// TwinCAT 3 PLC project Unbenannt1
// Title: Sample PackML_V2
// Company: Beckhoff Automation GmbH
// Author: Beckhoff Automation GmbH
// ProjectVersion: 3.0.3.0
// Description: Sample PackML_V2
// ProgramVersion: 3.1.4026.16
// libraries:
//   Tc2_MC2, * (Beckhoff Automation GmbH)
//   Tc2_Standard, * (Beckhoff Automation GmbH)
//   Tc2_System, * (Beckhoff Automation GmbH)
//   Tc2_Utilities, * (Beckhoff Automation GmbH)
//   Tc3_Analytics, * (Beckhoff Automation GmbH)
//   Tc3_Module, * (Beckhoff Automation GmbH)
//   Tc3_PackML_V2, * (Beckhoff Automation GmbH)
//   VisuDialogs, * (System)
// project tree:
//   DUTs/ E_PMLUserUnitMode.TcDUT, E_UnitName.TcDUT, ST_AxFunctions.TcDUT, ST_AxFunctionsAdmin.TcDUT, ST_ChangeIntoProduction.TcDUT, ST_AxFunctionsPTP.TcDUT, ST_UnitInfo.TcDUT
//   / GlobalTextList.TcGTLO, PlcTask.TcTTO, Visualization Manager.TcVMO (not stored)
//   GVLs/ GlobalVariables.TcGVL
//   POUs/General/ FB_AxisGeneral.TcPOU, FB_Cylinder.TcPOU, FB_Generic.TcPOU, FB_Velocity.TcPOU, FB_Visu.TcPOU, Ton_Break.TcPOU
//   POUs/ MAIN.TcPOU
//   POUs/Units/Conveyor/ FB_AxisMain.TcPOU
//   POUs/Units/Ejection/ FB_AxixEjection.TcPOU, FB_Ejector.TcPOU, FB_Sensor.TcPOU
//   POUs/Units/Machine/ FB_Machine.TcPOU
//   POUs/Units/Seperation/ FB_Seperation.TcPOU
//   Version/ Global_Version.TcGVL
//   VISUs/Templates/ VIS_TemplateCommand.TcVIS, VIS_TemplateKeys.TcVIS, VIS_TemplateMachine.TcVIS, VIS_TemplatePMLStateModel.TcVIS, VIS_TemplateToProduction.TcVIS
//   VISUs/ VIS_Main.TcVIS
// real-time tasks:
//   TASK PlcTask: cycle T#10ms, priority 20, ADS port 350
//   TASK PlcTask1: cycle T#10ms, priority 21, ADS port 351
//   TASK AnalyticsTask: cycle T#10ms, priority 1, ADS port 352
//   TASK AnalyticsTask_C1: cycle T#10ms, priority 22, ADS port 353
// motion (NC):
//   TASK NC-Task 1 SAF: cycle T#2ms, priority 4, ADS port 501
//   TASK NC-Task 1 SVB: cycle T#10ms, priority 8, ADS port 511
//   AXIS Axis 1 - Main Belt (id 1)
//     OtherSettings: AllowMotionCmdToSlave=true
//     encoder EncType=1
//     drive DrvType=5
//       TimeComp: TaskDelayCycles=1
//     controller CtrType=1
//       CtrPara: PriorControlFactor=1
//         Observer: BandWidth=20
//   AXIS Axis 2 - Metal Belt (id 2)
//     OtherSettings: AllowMotionCmdToSlave=true
//     encoder EncType=1
//     drive DrvType=5
//       TimeComp: TaskDelayCycles=1
//     controller CtrType=1
//       CtrPara: PriorControlFactor=1
//         Observer: BandWidth=20
//   AXIS Axis 3 - Plastic Belt (id 3)
//     OtherSettings: AllowMotionCmdToSlave=true
//     encoder EncType=1
//     drive DrvType=5
//       TimeComp: TaskDelayCycles=1
//     controller CtrType=1
//       CtrPara: PriorControlFactor=1
//         Observer: BandWidth=20
// variable links:
//   Unbenannt1/Unbenannt1 Instance <-> NC-Task 1 SAF/Axes/Axis 1 - Main Belt
//     PlcTask Inputs/GlobalVariables.AxisMain.NcToPlc <-> Outputs/ToPlc
//     PlcTask Outputs/GlobalVariables.AxisMain.PlcToNc <-> Inputs/FromPlc
//   Unbenannt1/Unbenannt1 Instance <-> NC-Task 1 SAF/Axes/Axis 2 - Metal Belt
//     PlcTask Inputs/GlobalVariables.AxisMetal.NcToPlc <-> Outputs/ToPlc
//     PlcTask Outputs/GlobalVariables.AxisMetal.PlcToNc <-> Inputs/FromPlc
//   Unbenannt1/Unbenannt1 Instance <-> NC-Task 1 SAF/Axes/Axis 3 - Plastic Belt
//     PlcTask Inputs/GlobalVariables.AxisPlastic.NcToPlc <-> Outputs/ToPlc
//     PlcTask Outputs/GlobalVariables.AxisPlastic.PlcToNc <-> Inputs/FromPlc
//   Unbenannt1/Unbenannt1 Instance <-> Unbenannt1/Unbenannt1 Instance
//     PlcTask Inputs/MAIN.fbMachine.fbEjectionMetal.bSensorEjection <-> PlcTask Outputs/MAIN.fbVisu.bMetalSensor
//     PlcTask Inputs/MAIN.fbMachine.fbEjectionMetal.fbCylinderEjection.bAtBasePos <-> PlcTask Outputs/MAIN.fbVisu.bMetalAtBase
//     PlcTask Inputs/MAIN.fbMachine.fbEjectionMetal.fbCylinderEjection.bAtWorkPos <-> PlcTask Outputs/MAIN.fbVisu.bMetalAtWork
//     PlcTask Inputs/MAIN.fbMachine.fbEjectionPlastic.bSensorEjection <-> PlcTask Outputs/MAIN.fbVisu.bPlasticSensor
//     PlcTask Inputs/MAIN.fbMachine.fbEjectionPlastic.fbCylinderEjection.bAtBasePos <-> PlcTask Outputs/MAIN.fbVisu.bPlasticAtBase
//     PlcTask Inputs/MAIN.fbMachine.fbEjectionPlastic.fbCylinderEjection.bAtWorkPos <-> PlcTask Outputs/MAIN.fbVisu.bPlasticAtWork
//     PlcTask Inputs/MAIN.fbMachine.fbSeperation.bSensorBarrier <-> PlcTask Outputs/MAIN.fbVisu.bBarrierSensor
//     PlcTask Inputs/MAIN.fbMachine.fbSeperation.fbCylinderBarrier.bAtBasePos <-> PlcTask Outputs/MAIN.fbVisu.bBarrierAtBase
//     PlcTask Inputs/MAIN.fbMachine.fbSeperation.fbCylinderBarrier.bAtWorkPos <-> PlcTask Outputs/MAIN.fbVisu.bBarrierAtWork
//     PlcTask Inputs/MAIN.fbMachine.fbSeperation.fbCylinderClamb.bAtBasePos <-> PlcTask Outputs/MAIN.fbVisu.bClampAtBase
//     PlcTask Inputs/MAIN.fbMachine.fbSeperation.fbCylinderClamb.bAtWorkPos <-> PlcTask Outputs/MAIN.fbVisu.bClampAtWork

CONFIGURATION Unbenannt1
    RESOURCE PLC ON TwinCAT3
        TASK PlcTask(INTERVAL := T#10ms, PRIORITY := 20);
        PROGRAM MAIN WITH PlcTask : MAIN;
    END_RESOURCE
END_CONFIGURATION

// ---- DUTs/E_PMLUserUnitMode.TcDUT
//Enumeration for User Modes
TYPE E_PMLUserUnitMode : (
	ePMLUnitMode_Service		:=  4,
	ePMLUnitMode_Usermode2		:=  5,
	ePMLUnitMode_Usermode3		:=  6,
	ePMLUnitMode_Usermode4		:=  7,
	ePMLUnitMode_Usermode5 		:=  8,
	ePMLUnitMode_Usermode6 		:=  9,
	ePMLUnitMode_Usermode7 		:=  10
) DINT;
END_TYPE

// ---- DUTs/E_UnitName.TcDUT
//Enumeration for Machineunits
TYPE E_UnitName :
(
	eMachine		:= 1,
	eSeperation		:= 2,
	eEjectorPlastic	:= 3,
	eAxisMain		:= 4,
	eEjectorMetal	:= 5,
	eSensorPlastic	:= 6,
	eAxisPlastic	:= 7,
	eSensorMetal	:= 8,
	eAxisMetal		:= 9
)DINT;
END_TYPE

// ---- DUTs/ST_AxFunctions.TcDUT
//structure includes structures with TC Motion functions
TYPE ST_AxFunctions :
STRUCT
	Admin				: ST_AxFunctionsAdmin;
	PTP					: ST_AxFunctionsPTP;
END_STRUCT
END_TYPE

// ---- DUTs/ST_AxFunctionsAdmin.TcDUT
//structure includes axisfunctions
TYPE ST_AxFunctionsAdmin :
STRUCT
	Power	: MC_Power;
	Reset	: MC_Reset;
END_STRUCT
END_TYPE

// ---- DUTs/ST_ChangeIntoProduction.TcDUT
//structure for a visu userwindow, to chnage into productionmode
TYPE ST_ChangeIntoProduction :
STRUCT
	bYes		: BOOL;
	bNo			: BOOL;
	bYesReset	: BOOL;
END_STRUCT
END_TYPE

// ---- DUTs/ST_AxFunctionsPTP.TcDUT
//structure includes point-to-point-functions
TYPE ST_AxFunctionsPTP :
STRUCT
	MoveVelocitiy		: MC_MoveVelocity;
	MoveAbsolute1		: MC_MoveAbsolute;
	MoveAbsolute2		: MC_MoveAbsolute;
	Stop				: MC_Stop;
	Halt				: MC_Halt;
END_STRUCT
END_TYPE

// ---- DUTs/ST_UnitInfo.TcDUT
//structure includes unit information
TYPE ST_UnitInfo :
STRUCT
	Name		: STRING;
	ActState	: E_PMLState;
	ActMode		: DINT;
END_STRUCT
END_TYPE

// ---- GVLs/GlobalVariables.TcGVL
VAR_GLOBAL
		AxisMain					: AXIS_REF;						//Main belt
		AxisPlastic					: AXIS_REF;						//Plastic belt
		AxisMetal					: AXIS_REF;						//Metal belt

		bAxisMainResetDone			: BOOL;							//True if main belt ressetting is finished 
		bPlasticEjectionResetDone	: BOOL;							//True if plasticejection ressetting is finished 
		bMetalEjectionResetDone		: BOOL;							//True if metalejection ressetting is finished 
		
		PackTags					: ST_PackMLv30;					//PackTags
		
		//analytics testing//2.1
		{attribute 'TcAnalytics'}
		nVisuProductCommand			: DINT:=1512000;							//Schedule products to produce

		bButtonProductionReq		: BOOL;							//TRUE when a mode change to PRODUCTION is requested
		stChangeIntoProduction		: ST_ChangeIntoProduction;		//Result of command box "Change to Production requested"

		aUnitInfo					: ARRAY [1..12] OF ST_UnitInfo;	//Array includes the states and modes of machineunits	
		aCaption					: ARRAY [1..12] OF STRING := ['F1','F2','F3','F4','F5','F6','F7','F8','F9','F10','F11','F12'];
		aKeyPressed					: ARRAY [1..12] OF BOOL;	
		
		
		uScheduleTime	 			: ULINT	:= 2 ;//for OEE 
		//analytics testing//2.1//3600000000000
		{attribute 'TcAnalytics'}			
		lScheduledTime 				: LINT	:= 3600000000000;//1 hours=1×60×60×1,000,000,000=3,600,000,000,000 nanoseconds
		
		//analytics testing//2.1
		{attribute 'TcAnalytics'}
		uDefectiveCount 			: ULINT	:= 0 ;//for OEE 
		
		//analytics testing//2.1
		{attribute 'TcAnalytics'}
		uTotalCount 				: ULINT	:= 0 ;//for OEE 
		
		//analytics testing//2.1
		{attribute 'TcAnalytics'}
		uPlasticCount 	 			: ULINT	:= 0 ;//for plastic items 
		
		//analytics testing//2.1
		{attribute 'TcAnalytics'}
		uMetalCount 	 			: ULINT	:= 0 ;//for metal items 
		
		//analytics testing//2.1
		{attribute 'TcAnalytics'}
		bScheduleDownTime 			: BOOL	:= FALSE ;//if under maintanance mode will be under this categories
		//analytics testing//2.1
		{attribute 'TcAnalytics'}
		bUnscheduleDownTime			: BOOL	:= FALSE ;//else if under manual mode or unknown will be under this categories
		
		//analytics testing//2.1
		{attribute 'TcAnalytics'}
		bProductionMode				: BOOL	:= FALSE ;//else if under manual mode or unknown will be under this categories
		
		//analytics testing//2.2
		{attribute 'TcAnalytics'}
		lStartTime 					: LWORD	:= 3600000000000 ;//Productivity internal
		//analytics testing//2.2
		{attribute 'TcAnalytics'}
		lStopTime 					: LWORD	:= 7200000000000 ;//Productivity internal
		
		//analytics testing//2.2
		{attribute 'TcAnalytics'}
		bConfigure 					: BOOL := TRUE;//Productivity internal
		
		{attribute 'TcAnalytics'}
		bReset	 					: BOOL := FALSE;//Productivity internal
		{attribute 'TcAnalytics'}
		bTest	 					: BOOL :=FALSE;//Productivity internal
END_VAR

// ---- Version/Global_Version.TcGVL
{attribute 'TcGenerated'}
{attribute 'no-analysis'}
{attribute 'linkalways'}
// This function has been automatically generated from the project information.
VAR_GLOBAL CONSTANT
	{attribute 'const_non_replaced'}
	stLibVersion_Sample_PackML_V2 : ST_LibVersion := (iMajor := 3, iMinor := 0, iBuild := 3, iRevision := 0, nFlags := 1, sVersion := '3.0.3.0');
END_VAR

// ---- POUs/MAIN.TcPOU
// Disclaimer
// 
// This publication contains statements about the suitability of our products for certain areas of application. These statements are based on typical features of our products. The examples shown in this publication are for demonstration purposes only. 
// The information provided herein should not be regarded as specific operation characteristics. It is incumbent on the customer to check and decide whether a product is suitable for use in a particular application. 
// We do not give any warranty that the source code which is made available with this publication is complete or accurate. 
//
// THE SAMPLE CODE CONTAINED IN THIS PUBLICATION IS PROVIDED “AS IS” WITHOUT WARRANTY OF ANY KIND, EITHER EXPRESSED, IMPLIED OR STATUTORY, INCLUDING WITHOUT LIMITATION, ANY WARRANTY WITH RESPECT TO NON-INFRINGEMENT, FREEDOM FROM PROPRIETARY RIGHTS OF THIRD PARTIES OR FITNESS FOR ANY PARTICULAR PURPOSE. 
// This publication may be changed from time to time without prior notice. No liability is assumed for errors and/or omissions. Our products are described in detail in our data sheets and documentations. Product-specific warnings and cautions must be observed. 
// For the latest version of our data sheets and documentations visit our website (www.beckhoff.de). 
//
// © Beckhoff Automation GmbH & Co. KG, 2022
// The reproduction, distribution and utilization of this document as well as the communication of its contents to others without express authorization is prohibited. Offenders will be held liable for the payment of damages. All rights reserved in the event of the grant of a patent, utility model or design.
PROGRAM MAIN
VAR_INPUT
	bExecuteComplete			: BOOL;									//Command Execute Complete, not defined
END_VAR
VAR
	UserModeCofig				: PML_UnitModeConfig;					//User can configure his own Mode
	
	fbMachine					: FB_Machine;							//Instance of FB_Machine
	bMachineStartedUp			: BOOL := FALSE;						//TRUE, when first PLC-Cycle finish

	fbVisu						: FB_Visu;								//Visualization
	
	fbTrigger					: F_TRIG;								//Trigger for resseting Counters

	fbLocalSystemTime			 : FB_LocalSystemTime;					//Get local Systemtime
	
	fbTriggerErrorMainAxis		: R_TRIG;								//Trigger for detecting Error on Mainaxis and write into PackTags
	fbTriggerErrorMetalAxis		: R_TRIG;								//Trigger for detecting Error on Metalaxis and write into PackTags
	fbTriggerErrorPlasticAxis	: R_TRIG;								//Trigger for detecting Error on Plasticaxis and write into PackTags
	
	nStateCommandCheck			: DINT;									//State to handle with statecommands
	//OEE UI
	todStart     				: TIME_OF_DAY:= TOD#00:00:00.000000000; // 8 AM
	//todStart     				: DT:=DT#2025-06-30-13:55:00;
	////todStart     				:  TIME := TIME#14H;
	//OEE UI
	todStop     				: TIME_OF_DAY:=TOD#09:00:00.000000000; // 5 PM
	//todStop     				: DT:=DT#2025-06-30-14:00:00;
	////todStop     				:  TIME := TIME#16H;

  	iLocalCount					: DINT;

	bTest1	:	BOOL;
	Test1	: TON;
END_VAR

//Configure Usermode 1
A_UnitModeConfig();

//Runs the first PLC-Cycle
IF fbMachine.bUndefinedDone AND NOT bMachineStartedUp THEN
	PackTags.Command.CntrlCmd	:= ePMLCommand_Abort;
	bMachineStartedUp			:= TRUE;
END_IF

M_SetPackTags();
M_SetPackTagsErrorWarning();

bButtonProductionReq := PackTags.Command.UnitMode = ePMLProtUnitMode_Production AND PackTags.Status.UnitModeCurrent <> PackTags.Command.UnitMode;

//Checking the Statecommands
CASE nStateCommandCheck OF
0:
	IF NOT (AxisMain.Status.Error OR AxisPlastic.Status.Error OR AxisMetal.Status.Error) THEN
		nStateCommandCheck:= 1;
	ELSE
		nStateCommandCheck:= 2;
	END_IF
1:
	IF PackTags.Command.CntrlCmd = ePMLCommand_Clear		
	  AND fbMachine.eState = ePMLState_Aborted	THEN
			fbMachine.eCommand	:= ePMLCommand_Clear;
	ELSIF PackTags.Command.CntrlCmd = ePMLCommand_Reset		
	  AND (fbMachine.eState = ePMLState_Stopped OR fbMachine.eState = ePMLState_Complete) THEN
			fbMachine.eCommand	:= ePMLCommand_Reset;
	ELSIF PackTags.Command.CntrlCmd = ePMLCommand_Start	
	  AND (fbMachine.eState = ePMLState_Idle OR (stPMLUnitModeConfiguration[fbMachine.eMode].aStateDisabled[ePMLState_Idle] AND fbMachine.eState = ePMLState_Stopped))
	  AND (NOT (PackTags.Command.Parameter[2].Value <= 0) OR NOT (fbMachine.eMode = 1))THEN
			fbMachine.eCommand	:= ePMLCommand_Start; 
	ELSIF PackTags.Command.CntrlCmd = ePMLCommand_Hold		
	  AND fbMachine.eState = ePMLState_Execute	
	  AND( fbMachine.eMode =  1 OR fbMachine.eMode =  4 OR fbMachine.eMode = 2)  THEN
			 fbMachine.eCommand	:= ePMLCommand_Hold;
	ELSIF PackTags.Command.CntrlCmd = ePMLCommand_Suspend	
	  AND fbMachine.eState = ePMLState_Execute	
	  AND (fbMachine.eMode = 4 OR fbMachine.eMode = 1)THEN
			 fbMachine.eCommand	:= ePMLCommand_Suspend;
	ELSIF PackTags.Command.CntrlCmd = ePMLCommand_Unhold	
	  AND fbMachine.eState = ePMLState_Held		THEN
			 fbMachine.eCommand	:= ePMLCommand_Unhold;
	ELSIF PackTags.Command.CntrlCmd = ePMLCommand_Unsuspend	
	  AND fbMachine.eState = ePMLState_Suspended	THEN
			 fbMachine.eCommand	:= ePMLCommand_Unsuspend;
	ELSIF PackTags.Command.CntrlCmd = ePMLCommand_Abort	THEN
			fbMachine.eCommand	:= ePMLCommand_Abort;
	ELSIF PackTags.Command.CntrlCmd = ePMLCommand_Stop	THEN
			fbMachine.eCommand	:= ePMLCommand_Stop;
	END_IF
	nStateCommandCheck:=0;
	
2:
	fbMachine.eCommand	:= ePMLCommand_Abort;
	IF fbMachine.eState = ePMLState_Aborted AND PackTags.Command.CntrlCmd = ePMLCommand_Clear THEN
		nStateCommandCheck:=1;
	END_IF
END_CASE

//
//Set the Packtags
M_SetPackTags();

//set the errors and warnings in Packtags
M_SetPackTagsErrorWarning();

//Call Visu
M_CallVisu();

//Call FB_Machine
fbMachine(eModeCommand:= PackTags.Command.UnitMode,  eMode => PackTags.Status.UnitModeCurrent, eState =>PackTags.Status.StateCurrent);

//for analytics conversion
lScheduledTime:= ULINT_TO_LINT(uScheduleTime*60*60*1000000000);
uTotalCount:= DINT_TO_ULINT(PackTags.Admin.ProdProcessedCount[1].Count);
uPlasticCount:= DINT_TO_ULINT(PackTags.Admin.ProdProcessedCount[3].Count);
uMetalCount:= DINT_TO_ULINT(PackTags.Admin.ProdProcessedCount[4].Count);

IF PackTags.Status.UnitModeCurrent = 1 THEN
	bProductionMode:= TRUE;
ELSE
	bProductionMode:= FALSE;
END_IF

//packml 2.2
// Convert to LWORD (100-ns ticks), then multiply
lStartTime := TO_LWORD(todStart) * 1000000;
lStopTime := TO_LWORD(todStop) * 1000000;

Test1(in:= bTest1,pt:= T#0.5S);
IF iLocalCount <> PackTags.Admin.ProdProcessedCount[1].Count THEN
	bTest:= TRUE;
	bTest1:= TRUE;
	iLocalCount := PackTags.Admin.ProdProcessedCount[1].Count;
ELSIF iLocalCount = PackTags.Admin.ProdProcessedCount[1].Count AND Test1.q THEN
	bTest:= FALSE;
	bTest1:= FALSE;
END_IF

ACTION A_UnitModeConfig:
UserModeCofig(
	eMode							:= ePMLUnitMode_Service, 
	bDisableClearing				:= TRUE, 
	bDisableStarting				:= TRUE, 
	bDisableSuspended				:= FALSE, 
	bDisableStopping				:= TRUE, 
	bDisableAborting				:= TRUE, 
	bDisableHolding					:= TRUE, 
	bDisableHeld					:= TRUE, 
	bDisableUnholding				:= TRUE, 
	bDisableSuspending				:= TRUE, 
	bDisableUnsuspending			:= TRUE, 
	bDisableResetting				:= TRUE, 
	bDisableIdle					:= TRUE, 
	bDisableCompleting				:= TRUE, 
	bDisableComplete				:= TRUE, 
	bEnableUnitModeChangeStopped	:= TRUE, 
	bEnableUnitModeChangeIdle		:= FALSE, 
	bEnableUnitModeChangeSuspended	:= FALSE, 
	bEnableUnitModeChangeExecute	:= FALSE, 
	bEnableUnitModeChangeAborted	:= TRUE, 
	bEnableUnitModeChangeHeld		:= FALSE, 
	bEnableUnitModeChangeComplete	:= FALSE, 
	bError							=> , 
	nErrorId						=> );
END_ACTION

METHOD M_CallVisu
VAR_INPUT
END_VAR
//Calling FB_Visu
fbVisu(
	fAxisVelo				:= PackTags.Command.Parameter[1].Value, 							
	bMainAxisMoves			:= AxisMain.Status.Moving, 
	bMetalAxisMoves			:= AxisMetal.Status.Moving, 
	bPlasticAxisMoves		:= AxisPlastic.Status.Moving, 
	bClampToWork			:= fbMachine.bClampToWork, 
	bBarrierToWork			:= fbMachine.bBarrierToWork, 
	bMetalToWork			:= fbMachine.bMetalToWork , 
	bPlasticToWork			:= fbMachine.bPlasticToWork ,
	bReset					:= ,
	aKeyPressed				:= aKeyPressed,
	aUnitInfo				:= aUnitInfo,
	fYClamp					=> , 
	fYBarrier				=> , 
	fYMetal					=> , 
	fYPlastic				=> , 
	bButtonPowerOut			=> , 
	bButtonMainFwOut		=> fbMachine.bButtonMainFw,  
	bButtonMetalFwOut		=> fbMachine.bButtonMetalFw, 
	bButtonPlasticFwOut		=> fbMachine.bButtonPlasticFw, 
	bButtonClampToWorkOut	=> fbMachine.bButtonClampToWork, 
	bButtonBarrierToWorkOut	=> fbMachine.bButtonBarrierToWork, 
	bButtonMetalToWorkOut	=> fbMachine.bButtonMetalToWork, 
	bButtonPlasticToWorkOut	=> fbMachine.bButtonPlasticToWork,
	bInvalidEntry			=> ,
	aCaption				=> aCaption,
	eModeVisu				=> ,
	eStateVisu				=> ,
	sUnitName				=> ,
	iFrameVisible			=> );
END_METHOD

METHOD M_SetPackTags
VAR_INPUT
END_VAR
VAR	
END_VAR
//***************************Writing Data into PackTags***************************
//Define the product metalbox 
PackTags.Command.Product[1].ProductID					:= 1;
PackTags.Command.Product[1].ProcessVariables[1].ID		:= 1;
PackTags.Command.Product[1].ProcessVariables[1].Name	:= 'CylinderPressureMetal';
PackTags.Command.Product[1].ProcessVariables[1].Unit	:= 'Bar';
PackTags.Command.Product[1].ProcessVariables[1].Value	:= 5;
(*Thre are no useful Ingrediens for Metalboxes in this Machine*)

//Define the product plasticbox
PackTags.Command.Product[2].ProductID					:= 2;
PackTags.Command.Product[2].ProcessVariables[1].ID		:= 2;
PackTags.Command.Product[2].ProcessVariables[1].Name	:= 'CylinderPressurePlastic';
PackTags.Command.Product[2].ProcessVariables[1].Unit	:= 'Bar';
PackTags.Command.Product[2].ProcessVariables[1].Value	:= 3;
(*Thre are no useful Ingrediens for Plasticboxes in this Machine*)

//Parameters for the production, here set the velocity from MainBelt
PackTags.Command.Parameter[1].ID				:= 3;
PackTags.Command.Parameter[1].Name				:= 'MainBeltVelo';
PackTags.Command.Parameter[1].Unit				:= 'mm/s';
PackTags.Command.Parameter[1].Value				:= 100.0;

//Number of producing products
PackTags.Command.Parameter[2].ID				:= 4;
PackTags.Command.Parameter[2].Name				:= 'Quantity';
PackTags.Command.Parameter[2].Unit				:= 'Box';

//Parameters for the production, here set the velocity from MetalBelt
PackTags.Command.Parameter[3].ID				:= 5;
PackTags.Command.Parameter[3].Name				:= 'MetalBeltVelo';
PackTags.Command.Parameter[3].Unit				:= 'mm/s';
PackTags.Command.Parameter[3].Value				:= 100.0;

//Parameters for the production, here set the velocity from PlasticBelt
PackTags.Command.Parameter[4].ID				:= 6;
PackTags.Command.Parameter[4].Name				:= 'PlasticBeltVelo';
PackTags.Command.Parameter[4].Unit				:= 'mm/s';
PackTags.Command.Parameter[4].Value				:= 100.0;

//Parameters for the production, here get the velocity from PlasticBelt
PackTags.Status.Parameter[1].ID					:= 7;
PackTags.Status.Parameter[1].Name				:= 'MainBeltVelo';
PackTags.Status.Parameter[1].Unit				:= 'mm/s';
PackTags.Status.Parameter[1].Value				:= LREAL_TO_REAL(AxisMain.NcToPlc.ActVelo);

//Parameters for the production, here get the velocity from PlasticBelt
PackTags.Status.Parameter[2].ID					:= 8;
PackTags.Status.Parameter[2].Name				:= 'MetalBeltVelo';
PackTags.Status.Parameter[2].Unit				:= 'mm/s';
PackTags.Status.Parameter[2].Value				:=  LREAL_TO_REAL(AxisMetal.NcToPlc.ActVelo);

//Parameters for the production, here get the velocity from PlasticBelt
PackTags.Status.Parameter[3].ID					:= 9;
PackTags.Status.Parameter[3].Name				:= 'PlasticBeltVelo';
PackTags.Status.Parameter[3].Unit				:= 'mm/s';
PackTags.Status.Parameter[3].Value				:=  LREAL_TO_REAL(AxisPlastic.NcToPlc.ActVelo);

//Countig produced boxes, see FB_Ejection
PackTags.Admin.ProdProcessedCount[1].ID			:= 1;
PackTags.Admin.ProdProcessedCount[1].Name		:= 'BoxfinishEjectionAll';
PackTags.Admin.ProdProcessedCount[1].Unit		:= 'Box';

//Countig produced boxes, see FB_Seperation
PackTags.Admin.ProdProcessedCount[2].ID			:= 2;
PackTags.Admin.ProdProcessedCount[2].Name		:= 'BoxfinishSeperation';
PackTags.Admin.ProdProcessedCount[2].Unit		:= 'Boxes';

//Countig produced boxes, see FB_EjectionPlastic
PackTags.Admin.ProdProcessedCount[3].ID			:= 3;
PackTags.Admin.ProdProcessedCount[3].Name		:= 'BoxFinishPlastic';
PackTags.Admin.ProdProcessedCount[3].Unit		:= 'Boxes';

//Countig produced boxes, see FB_EjectionMetal
PackTags.Admin.ProdProcessedCount[4].ID			:= 4;
PackTags.Admin.ProdProcessedCount[4].Name		:= 'BoxFinishMetal';
PackTags.Admin.ProdProcessedCount[4].Unit		:= 'Boxes';

//Write the actual state and mode into the PackTags
PackTags.Status.StateCurrent					:= fbMachine.eState;
PackTags.Status.UnitModeCurrent					:= fbMachine.eMode;
PackTags.Status.StateRequested					:= fbMachine.eCommand;
PackTags.Status.UnitModeRequested				:= fbMachine.eModeCommand;
PackTags.Status.StateChangeInProcess			:= PackTags.Status.StateCurrent <> PackTags.Status.StateRequested;
PackTags.Status.UnitModeChangeInProcess			:= PackTags.Status.UnitModeCurrent <> PackTags.Status.UnitModeRequested;

//Write actual time and date in PackTags
fbLocalSystemTime(sNetID:= '', bEnable := TRUE);
PackTags.Admin.PlcDateTime[0]	:= fbLocalSystemTime.systemTime.wYear;
PackTags.Admin.PlcDateTime[1]	:= fbLocalSystemTime.systemTime.wMonth;
PackTags.Admin.PlcDateTime[2]	:= fbLocalSystemTime.systemTime.wDay;
PackTags.Admin.PlcDateTime[3]	:= fbLocalSystemTime.systemTime.wHour;
PackTags.Admin.PlcDateTime[4]	:= fbLocalSystemTime.systemTime.wMinute;
PackTags.Admin.PlcDateTime[5]	:= fbLocalSystemTime.systemTime.wSecond;
PackTags.Admin.PlcDateTime[6]	:= fbLocalSystemTime.systemTime.wMilliseconds;


//Set the productcounter to 0, when the production command is completed
fbTrigger(CLK:= (fbMachine.eState = ePMLState_Complete));
IF fbTrigger.Q OR stChangeIntoProduction.bYesReset THEN
	PackTags.Admin.ProdProcessedCount[1].Count	:= 0;
	PackTags.Admin.ProdProcessedCount[2].Count	:= 0;
	PackTags.Admin.ProdProcessedCount[3].Count	:= 0;
	PackTags.Admin.ProdProcessedCount[4].Count	:= 0;
	PackTags.Command.Parameter[2].Value			:= 0;
	nVisuProductCommand							:= 0;
END_IF
END_METHOD

METHOD M_SetPackTagsErrorWarning
VAR_INPUT
END_VAR
//====================Error and Warnig setting========================
//Warnings
PackTags.Admin.Warning[1].Message	:= 'Invalid Production Command, command Products must be higher than 0';
PackTags.Admin.Warning[1].ID 		:= 1;

PackTags.Admin.Warning[2].Message	:= 'Invalid Mode Command, please try anothereone';
PackTags.Admin.Warning[2].ID		:= 2;

//Errors
PackTags.Admin.Alarm[1].Message		:= 'Error on Main Axis';
PackTags.Admin.Alarm[1].ID			:= 1;

PackTags.Admin.Alarm[2].Message		:= 'Error on Metal Axis';
PackTags.Admin.Alarm[2].ID			:= 2;

PackTags.Admin.Alarm[3].Message		:= 'Error on Plastic Belt';
PackTags.Admin.Alarm[3].ID			:= 3;

//====================Error and Warnig handling========================
//warning for invalid production command
IF PackTags.Status.UnitModeCurrent = ePMLProtUnitMode_Production AND PackTags.Status.StateCurrent = ePMLState_Idle AND PackTags.Command.CntrlCmd = ePMLCommand_Start AND PackTags.Command.Parameter[2].Value <= 0 THEN
	PackTags.Admin.Warning[1].Trigger :=TRUE;
ELSE
	PackTags.Admin.Warning[1].Trigger :=FALSE;
END_IF

//warning for invalid mode command
IF fbMachine.bInvalidModeCommandOut THEN
	PackTags.Admin.Warning[2].Trigger :=TRUE;
ELSE 
	PackTags.Admin.Warning[2].Trigger :=FALSE;
END_IF

//===============Axis Errors===================
//Main Axis
fbTriggerErrorMainAxis(CLK:= AxisMain.Status.Error);
IF fbTriggerErrorMainAxis.Q THEN
	PackTags.Admin.Alarm[1].DateTime	:= PackTags.Admin.PlcDateTime;
END_IF
IF AxisMain.Status.Error THEN
	PackTags.Admin.Alarm[1].Trigger		:= TRUE;
	PackTags.Admin.Alarm[1].Value		:= UDINT_TO_DINT(AxisMain.Status.ErrorID);
ELSE
	PackTags.Admin.Alarm[1].Trigger		:= FALSE;
	MEMSET(ADR(PackTags.Admin.Alarm[1].DateTime),0,SIZEOF(PackTags.Admin.Alarm[1].DateTime));
END_IF

//Metal Axis
fbTriggerErrorMetalAxis(CLK:= AxisMetal.Status.Error);
IF fbTriggerErrorMetalAxis.Q THEN
	PackTags.Admin.Alarm[2].DateTime	:= PackTags.Admin.PlcDateTime;
END_IF
IF AxisMetal.Status.Error THEN
	PackTags.Admin.Alarm[2].Trigger		:= TRUE;
	PackTags.Admin.Alarm[2].Value		:= UDINT_TO_DINT(AxisMetal.Status.ErrorID);
ELSE
	PackTags.Admin.Alarm[2].Trigger		:= FALSE;
	MEMSET(ADR(PackTags.Admin.Alarm[2].DateTime),0,SIZEOF(PackTags.Admin.Alarm[2].DateTime));
END_IF

//Plastic Axis
fbTriggerErrorPlasticAxis(CLK:= AxisPlastic.Status.Error);
IF fbTriggerErrorPlasticAxis.Q THEN
	PackTags.Admin.Alarm[3].DateTime	:= PackTags.Admin.PlcDateTime;	
END_IF
IF AxisPlastic.Status.Error THEN
	PackTags.Admin.Alarm[3].Trigger		:= TRUE;
	PackTags.Admin.Alarm[3].Value		:= UDINT_TO_DINT(AxisPlastic.Status.ErrorID);
ELSE
	PackTags.Admin.Alarm[3].Trigger		:= FALSE;
	MEMSET(ADR(PackTags.Admin.Alarm[3].DateTime),0,SIZEOF(PackTags.Admin.Alarm[3].DateTime));
END_IF
END_METHOD

END_PROGRAM

// ---- POUs/Units/Machine/FB_Machine.TcPOU
FUNCTION_BLOCK FB_Machine EXTENDS FB_Generic
VAR_INPUT
	bButtonMainFw			: BOOL; 
	bButtonMetalFw			: BOOL; 
	bButtonPlasticFw		: BOOL; 
	bButtonClampToWork		: BOOL; 
	bButtonBarrierToWork	: BOOL; 
	bButtonMetalToWork		: BOOL; 
	bButtonPlasticToWork	: BOOL;
END_VAR
VAR_OUTPUT
	bClampToWork			: BOOL; 
	bBarrierToWork			: BOOL;
	bMetalToWork			: BOOL;
	bPlasticToWork			: BOOL;
END_VAR
VAR	
	fbAxisMain			: FB_AxisMain;							//Main Belt Unit			
	fbSeperation		: FB_Seperation;						//Separating unit	
	fbEjectionPlastic	: FB_Ejector;							//Unit that sorts plastic boxes
	fbEjectionMetal		: FB_Ejector;							//Unit that sorts metal boxes
	
	stSubModuleInfo		: ARRAY [1..4] OF ST_PMLSubUnitInfo;	//Informations about the Subunits

	fbVelocity			: FB_Velocity;							//calculate the actual and average velocity
END_VAR

//=======================Main Belt=======================
fbAxisMain(		
	Axis				:= AxisMain,
	eModeCommand		:= eModeCommand,
	eCommand 			:= eCommand,
	bMoveFw				:= bButtonMainFw,
	fConveyorLenght		:= 1300.0,
	fConveyorVelo		:= PackTags.Command.Parameter[1].Value,
	eMode 				=> ,
	eState				=> stSubModuleInfo[1].eState,
	bResettingDone		=> bAxisMainResetDone);				
	
stSubModuleInfo[1].Active		:= TRUE;

//=======================Separating Modul=======================
fbSeperation(	
	eModeCommand		:= eModeCommand,
	eCommand 			:= eCommand,
	bMoveClambCylinder	:= bButtonClampToWork,
	bMoveBarrierCylinder:= bButtonBarrierToWork,
	eMode 				=> ,
	eState				=> stSubModuleInfo[2].eState,
	bMoveToWorkClambHw	=> bClampToWork,
	bMoveToWorkBarrierHw=> bBarrierToWork);

stSubModuleInfo[2].Active		:= TRUE;

//=======================Plastic Ejection=======================
fbEjectionPlastic(	
	Axis			:= AxisPlastic,
	eModeCommand	:= eModeCommand,
	eCommand 		:= eCommand,
	bMoveBeltFw		:= bButtonPlasticFw,
	bMoveCylinder	:= bButtonPlasticToWork,
	eMode 			=> ,
	eState			=>  stSubModuleInfo[3].eState,
	bResetDone		=> bPlasticEjectionResetDone,
	nCounterProduct	=> PackTags.Admin.ProdProcessedCount[3].Count,
	bMoveToWork		=> bPlasticToWork);			

stSubModuleInfo[3].Active			:= TRUE;

//=======================Metal Ejection=======================
fbEjectionMetal(	
	Axis			:= AxisMetal,
	eModeCommand	:= eModeCommand,
	eCommand		:= eCommand,
	bMoveBeltFw		:= bButtonMetalFw,
	bMoveCylinder	:= bButtonMetalToWork,
	eMode			=> ,
	eState			=> stSubModuleInfo[4].eState,
	bResetDone		=> bMetalEjectionResetDone,
	nCounterProduct	=> PackTags.Admin.ProdProcessedCount[4].Count,
	bMoveToWork		=> bMetalToWork);			

stSubModuleInfo[4].Active	:= TRUE;

//The fbStateMachine from FB_Machine gets the Information about the states and activity from the subunits
fbStateMachine.stSubUnitInfoRef.ArraySize		:= SIZEOF(stSubModuleInfo);
fbStateMachine.stSubUnitInfoRef.NoOfSubUnits	:= 4;
fbStateMachine.stSubUnitInfoRef.pArray			:= ADR(stSubModuleInfo);

IF  fbAxisMain.bUndefinedDone AND fbEjectionMetal.bUndefinedDone AND fbEjectionPlastic.bUndefinedDone AND fbSeperation.bUndefinedDone THEN
	bUndefinedDone := TRUE;
END_IF

//Set unit information 
M_SetUnitInfo();

fbVelocity(nActQuantity:= PackTags.Admin.ProdProcessedCount[1].Count, fActVelocity=> PackTags.Status.CurMachineSpeed, fAverageVelo=> PackTags.Status.MachineSpeed);

SUPER^();

METHOD M_SetUnitInfo
VAR_INPUT
END_VAR
aUnitInfo[eMachine].Name			:= 'fbMachine';
aUnitInfo[eMachine].ActMode			:= eMode;
aUnitInfo[eMachine].ActState		:= eState;

aUnitInfo[eSeperation].Name			:= 'fbSeperation';
aUnitInfo[eSeperation].ActMode		:= fbSeperation.eMode;
aUnitInfo[eSeperation].ActState		:= fbSeperation.eState;


aUnitInfo[eEjectorPlastic].Name		:= 'fbEjectorPlastic';
aUnitInfo[eEjectorPlastic].ActMode	:= fbEjectionPlastic.eMode;
aUnitInfo[eEjectorPlastic].ActState	:= fbEjectionPlastic.eState;


aUnitInfo[eAxisMain].Name			:= 'fbAxisMain';
aUnitInfo[eAxisMain].ActMode		:= fbAxisMain.eMode;
aUnitInfo[eAxisMain].ActState		:= fbAxisMain.eState;


aUnitInfo[eEjectorMetal].Name		:= 'fbEjectorMetal';
aUnitInfo[eEjectorMetal].ActMode	:= fbEjectionMetal.eMode;
aUnitInfo[eEjectorMetal].ActState	:= fbEjectionMetal.eState;


aUnitInfo[eSensorPlastic].Name		:= 'fbSensorPlastic';
aUnitInfo[eSensorPlastic].ActMode	:= fbEjectionPlastic.eModeSensor;
aUnitInfo[eSensorPlastic].ActState	:= fbEjectionPlastic.eStateSesnor;


aUnitInfo[eAxisPlastic].Name		:= 'fbAxisplastic';
aUnitInfo[eAxisPlastic].ActMode		:= fbEjectionPlastic.eModeAxis;
aUnitInfo[eAxisPlastic].ActState	:= fbEjectionPlastic.eStateAxis;

aUnitInfo[eSensorMetal].Name		:= 'fbSensorMetal';
aUnitInfo[eSensorMetal].ActMode		:= fbEjectionMetal.eModeSensor;
aUnitInfo[eSensorMetal].ActState	:= fbEjectionMetal.eStateSesnor;


aUnitInfo[eAxisMetal].Name			:= 'fbAxisMetal';
aUnitInfo[eAxisMetal].ActMode		:= fbEjectionMetal.eModeAxis;
aUnitInfo[eAxisMetal].ActState		:= fbEjectionMetal.eStateAxis;
END_METHOD

END_FUNCTION_BLOCK

// ---- POUs/General/FB_Generic.TcPOU
//the functionblock FB_Generick is transmitted to every machineunit
FUNCTION_BLOCK FB_Generic IMPLEMENTS ITF_UnitState
VAR_INPUT
	eModeCommand			: DINT;									//Mode from superior Unit
	eCommand				: E_PMLCommand := ePMLCommand_Abort;	//Command for a new state from superior unit
END_VAR
VAR_OUTPUT
	eMode					: DINT;									//Actual mode of the Unit
	eState					: E_PMLState (*:= ePMLState_Aborted*) ;	//Actual state of the Unit
	bUndefinedDone			: BOOL;									//When the SPS is started, the first state is Undefiend. bUndefined is TRUE, when the method Undefined has succesful finished
	bInvalidModeCommandOut	: BOOL;
	bChangeIntoProduction	: BOOL;
END_VAR
VAR
	fbUnitModeManager		: PML_UnitModeManager;					//The PML_UnitModeManager manage the Modechanges
	fbStateMachine 			: PML_StateMachine;						//The PML_StateMachine mangae the Statechanges
	
	nStateModeChange		: INT	:= 0;							//Variable to handle the modechange
	nLastState				: E_PMLState;							//Variable to store last state
END_VAR

CASE nStateModeChange OF
0:
	//Waiting for user request
	bChangeIntoProduction:= FALSE;
	IF  bButtonProductionReq AND (PackTags.Command.UnitMode = ePMLProtUnitMode_Production) AND (PackTags.Status.UnitModeCurrent = ePMLProtUnitMode_Invalid) THEN
			nStateModeChange	:= 1;
	ELSIF  PackTags.Command.UnitModeChangeRequest AND (PackTags.Command.UnitMode <> ePMLProtUnitMode_Production) THEN
			nStateModeChange	:= 1;
	ELSIF  bButtonProductionReq AND (PackTags.Command.UnitMode = ePMLProtUnitMode_Production) AND (PackTags.Status.UnitModeCurrent <> ePMLProtUnitMode_Production) THEN
			nStateModeChange	:= 3;
	END_IF
1:
	//Starting UnitModeManager 
	fbUnitModeManager.bExecute				:= TRUE;
	fbUnitModeManager.eModeCommand			:= eModeCommand;
	PackTags.Status.UnitModeChangeInProcess	:= TRUE;

	IF fbUnitModeManager.bDone THEN
		fbUnitModeManager.bExecute	:= FALSE;
		bInvalidModeCommandOut		:= FALSE;
		nStateModeChange			:= 0;
		bChangeIntoProduction		:= FALSE;
		PackTags.Status.UnitModeChangeInProcess	:= FALSE;
	ELSIF fbUnitModeManager.bError THEN
		bInvalidModeCommandOut		:= TRUE;
		fbUnitModeManager.bExecute	:= FALSE;
		nLastState					:= PackTags.Status.StateCurrent;
		nLastState					:= PackTags.Status.StateCurrent;
		nStateModeChange			:= 2;
		bChangeIntoProduction		:= FALSE;
		PackTags.Status.UnitModeChangeInProcess	:= FALSE;
	END_IF
2:
	//ErrorHanddling
	IF  PackTags.Command.UnitModeChangeRequest THEN
		nStateModeChange:=0;
		bInvalidModeCommandOut		:= FALSE;
	ELSIF nLastState<> PackTags.Status.StateCurrent THEN
		bInvalidModeCommandOut		:= FALSE;
	END_IF
	
3:
	//state to check, if command 'Porduction' is valid
	IF (PackTags.Status.StateCurrent = ePMLState_Aborted OR PackTags.Status.StateCurrent = ePMLState_Stopped OR PackTags.Status.StateCurrent = ePMLState_Idle) THEN
		bChangeIntoProduction		:= TRUE;
		IF stChangeIntoProduction.bYes OR stChangeIntoProduction.bYesReset THEN
			nStateModeChange			:= 1;		
		ELSIF stChangeIntoProduction.bNo THEN
			nStateModeChange			:= 0;
		END_IF
	ELSE
		nStateModeChange:= 2;
		bInvalidModeCommandOut		:= TRUE;
		nLastState					:= PackTags.Status.StateCurrent;
	END_IF
END_CASE


fbUnitModeManager(									
	eState			:= eState,
	eModeStatus		=> eMode,
	bDone			=> ,
	bError			=> ,
	nErrorId		=> );


IF fbUnitModeManager.eModeStatus <>  0 THEN
	//Calling the StateMachine, when there is a valid Mode
	fbStateMachine(
		eMode				:= eMode, 				
		eCommand			:= eCommand,			
		stSubUnitInfoRef	:= ,
		stOptions			:= , 
		eState				=> eState, 				
		bError				=> , 
		nErrorID			=> );
END_IF

//One of the methods is executing  by the actual state
CASE eState OF
	ePMLState_Undefined:
		M_Undefined();
	ePMLState_Clearing:
		M_Clearing();
	ePMLState_Stopped:
		M_Stopped();
	ePMLState_Starting:
		M_Starting();
	ePMLState_Idle:
		M_Idle();
	ePMLState_Suspended:
		M_Suspended();
	ePMLState_Execute:
		M_Execute();
	ePMLState_Stopping:
		M_Stopping();
	ePMLState_Aborting:
		M_Aborting();
	ePMLState_Aborted:
		M_Aborted();
	ePMLState_Holding:
		M_Holding();
	ePMLState_Held:
		M_Held();
	ePMLState_Unholding:
		M_Unholding();
	ePMLState_Suspending:
		M_Suspending();
	ePMLState_Unsuspending:
		M_Unsuspending();
	ePMLState_Resetting:
		M_Resetting();
	ePMLState_Completing:
		M_Completing();
	ePMLState_Complete:
		M_Complete();
END_CASE

{attribute 'object_name' := 'M_Aborted'}
METHOD M_Aborted
END_METHOD

{attribute 'object_name' := 'M_Aborting'}
METHOD M_Aborting
M_StateComplete();
END_METHOD

{attribute 'object_name' := 'M_Clearing'}
METHOD M_Clearing
M_StateComplete();
END_METHOD

{attribute 'object_name' := 'M_Complete'}
METHOD M_Complete
END_METHOD

{attribute 'object_name' := 'M_Completing'}
METHOD M_Completing
M_StateComplete();
END_METHOD

{attribute 'object_name' := 'M_Execute'}
METHOD M_Execute
M_StateComplete();
END_METHOD

{attribute 'object_name' := 'M_Held'}
METHOD M_Held
END_METHOD

{attribute 'object_name' := 'M_Holding'}
METHOD M_Holding
M_StateComplete();
END_METHOD

{attribute 'object_name' := 'M_Idle'}
METHOD M_Idle
END_METHOD

{attribute 'object_name' := 'M_Resetting'}
METHOD M_Resetting
M_StateComplete();
END_METHOD

{attribute 'object_name' := 'M_Starting'}
METHOD M_Starting
M_StateComplete();
END_METHOD

{attribute 'object_name' := 'M_StateComplete'}
METHOD M_StateComplete
//the actual state is completed
fbStateMachine.M_StateComplete();
END_METHOD

{attribute 'object_name' := 'M_Stopped'}
METHOD M_Stopped
END_METHOD

{attribute 'object_name' := 'M_Stopping'}
METHOD M_Stopping
M_StateComplete();
END_METHOD

{attribute 'object_name' := 'M_Suspended'}
METHOD M_Suspended
END_METHOD

{attribute 'object_name' := 'M_Suspending'}
METHOD M_Suspending
M_StateComplete();
END_METHOD

{attribute 'object_name' := 'M_Undefined'}
METHOD M_Undefined
END_METHOD

{attribute 'object_name' := 'M_Unholding'}
METHOD M_Unholding
M_StateComplete();
END_METHOD

{attribute 'object_name' := 'M_Unsuspending'}
METHOD M_Unsuspending
M_StateComplete();
END_METHOD

END_FUNCTION_BLOCK

// ---- POUs/Units/Conveyor/FB_AxisMain.TcPOU
FUNCTION_BLOCK FB_AxisMain EXTENDS FB_AxisGeneral

//Call the FB_Axis_General and hand over the Axis References
SUPER^(Axis := Axis);

{attribute 'object_name' := 'M_Completing'}
METHOD M_Completing
CASE fbUnitModeManager.eModeStatus OF
	ePMLProtUnitMode_Production:
		//The main belt run on for a box length
		stAxis.PTP.MoveAbsolute1.Velocity		:= fConveyorVelo;
		stAxis.PTP.MoveAbsolute1.Acceleration	:= 0;
		stAxis.PTP.MoveAbsolute1.BufferMode		:= MC_Aborting;
		stAxis.PTP.MoveAbsolute1.Deceleration	:= 0;
		stAxis.PTP.MoveAbsolute1.Execute		:= TRUE;
		stAxis.PTP.MoveAbsolute1.Jerk			:= 0;
		stAxis.PTP.MoveAbsolute1.Position		:= (Axis.NcToPlc.ActPos + 200);
		IF stAxis.PTP.MoveAbsolute1.Done  THEN
			stAxis.PTP.MoveAbsolute1.Execute	:= FALSE;
			SUPER^.M_Completing();
		END_IF
END_CASE
END_METHOD

{attribute 'object_name' := 'M_Execute'}
METHOD M_Execute
CASE fbUnitModeManager.eModeStatus OF
	ePMLProtUnitMode_Production:		//Productionmode
		//Move the axis with const. velocity
		stAxis.PTP.MoveVelocitiy.Acceleration		:= 0;
		stAxis.PTP.MoveVelocitiy.BufferMode		:= MC_Aborting;
		stAxis.PTP.MoveVelocitiy.Deceleration		:= 0;
		stAxis.PTP.MoveVelocitiy.Direction			:= MC_Positive_Direction;
		stAxis.PTP.MoveVelocitiy.Execute			:= TRUE;
		stAxis.PTP.MoveVelocitiy.Jerk				:= 0;
		stAxis.PTP.MoveVelocitiy.Velocity			:= PackTags.Command.Parameter[1].Value;
		
		//If the output target is reached, the machine stops and chnage the state
		IF  REAL_TO_DINT(PackTags.Command.Parameter[2].Value) <= PackTags.Admin.ProdProcessedCount[1].Count  THEN
			stAxis.PTP.MoveVelocitiy.Execute	:= FALSE;
			stAxis.PTP.Stop.Deceleration		:= 0;
			stAxis.PTP.Stop.Execute				:= TRUE;
			stAxis.PTP.Stop.Jerk				:= 0;
			IF stAxis.PTP.Stop.Done AND PackTags.Status.StateCurrent = ePMLState_Execute  THEN
				stAxis.PTP.Stop.Execute			:= FALSE;
				M_StateComplete();
			END_IF
		END_IF
		 
	ePMLProtUnitMode_Maintenance:		//Mantainancemode
		stAxis.PTP.Stop.Deceleration				:= 0;
		stAxis.PTP.Stop.Execute						:= TRUE;
		stAxis.PTP.Stop.Jerk						:= 0;

	ePMLProtUnitMode_Manual:		//Manualmode
		//Call FB_AxisGeneral
		SUPER^.M_Execute();
		
	ePMLUnitMode_Service:		//UserMode
		//Not defined
END_CASE
END_METHOD

{attribute 'object_name' := 'M_Holding'}
METHOD M_Holding
CASE fbUnitModeManager.eModeStatus OF
	ePMLProtUnitMode_Production:		//Production
		//Move the half lenght of the belt, to bring every box to the destination
		stAxis.PTP.MoveVelocitiy.Execute		:= FALSE;
		stAxis.PTP.MoveAbsolute1.Acceleration	:= 0;
		stAxis.PTP.MoveAbsolute1.BufferMode		:= MC_Aborting;
		stAxis.PTP.MoveAbsolute1.Deceleration	:= 0;
		stAxis.PTP.MoveAbsolute1.Execute		:= TRUE;
		stAxis.PTP.MoveAbsolute1.Jerk			:= 0;
		stAxis.PTP.MoveAbsolute1.Velocity		:= PackTags.Command.Parameter[1].Value;
		stAxis.PTP.MoveAbsolute1.Position		:= (AxisMain.NcToPlc.ActPos + fConveyorLenght); //Drive actual Position + Length of Conveyor
		
		IF stAxis.PTP.MoveAbsolute1.Done THEN
			stAxis.PTP.MoveAbsolute1.Execute	:= FALSE;
			M_StateComplete();
		END_IF
								
	ePMLProtUnitMode_Maintenance:		//Mantainance
		M_StateComplete();				
END_CASE
END_METHOD

{attribute 'object_name' := 'M_Resetting'}
METHOD M_Resetting
CASE fbStateMachine.eMode OF
		
	ePMLProtUnitMode_Production:
		CASE iStateResetting OF
			0:		
				//SW-Enable the axis
				bResettingDone										:= FALSE;
				stAxis.Admin.Power.BufferMode			:= MC_Aborting;
				stAxis.Admin.Power.Enable				:= TRUE;
				stAxis.Admin.Power.Enable_Negative		:= TRUE;
				stAxis.Admin.Power.Enable_Positive		:= TRUE;
				stAxis.Admin.Power.Override				:= 100.0;
				IF stAxis.Admin.Power.Status THEN
					iStateResetting	:= 1;
				END_IF
				
			1:
				//Take away all Move-Commands
				stAxis.PTP.Halt.Execute					:= FALSE;
				stAxis.PTP.MoveAbsolute1.Execute		:= FALSE;
				stAxis.PTP.MoveAbsolute2.Execute		:= FALSE;
				stAxis.PTP.MoveVelocitiy.Execute		:= FALSE;
				stAxis.PTP.Stop.Execute					:= FALSE;
				IF AxisMetal.Status.NotMoving AND AxisPlastic.Status.NotMoving AND bPlasticEjectionResetDone AND bMetalEjectionResetDone AND NOT Axis.Status.HasJob THEN
					iStateResetting									:= 2;
				END_IF
			
			2:
				//Move the axis for one conveyorroatation
				stAxis.PTP.MoveAbsolute1.Acceleration	:= 0;
				stAxis.PTP.MoveAbsolute1.BufferMode		:= MC_BlendingPrevious;
				stAxis.PTP.MoveAbsolute1.Deceleration	:= 0;
				stAxis.PTP.MoveAbsolute1.Execute		:= TRUE;
				stAxis.PTP.MoveAbsolute1.Jerk			:= 0;
				stAxis.PTP.MoveAbsolute1.Velocity		:= fConveyorVelo;
				stAxis.PTP.MoveAbsolute1.Position		:= (AxisMain.NcToPlc.ActPos + fConveyorLenght); //Drive actual Position + Length of Conveyor
			IF stAxis.PTP.MoveAbsolute1.Done THEN
				bResettingDone				:= TRUE;
				stAxis.PTP.MoveAbsolute1.Execute		:= FALSE;
				M_StateComplete();
			END_IF
		END_CASE

	ePMLProtUnitMode_Maintenance:
		M_StateComplete();

	ePMLProtUnitMode_Manual:	
		SUPER^.M_Resetting();

	ePMLUnitMode_Service:
		M_StateComplete();
END_CASE
END_METHOD

{attribute 'object_name' := 'M_Suspending'}
METHOD M_Suspending
CASE fbUnitModeManager.eModeStatus OF
	ePMLProtUnitMode_Production:		
		//The main belt run on for the half beltlength
		stAxis.PTP.MoveVelocitiy.Execute		:= FALSE;
		stAxis.PTP.MoveAbsolute1.Acceleration	:= 0;
		stAxis.PTP.MoveAbsolute1.BufferMode		:= MC_Aborting;
		stAxis.PTP.MoveAbsolute1.Deceleration	:= 0;
		stAxis.PTP.MoveAbsolute1.Execute		:= TRUE;		
		stAxis.PTP.MoveAbsolute1.Jerk			:= 0;
		stAxis.PTP.MoveAbsolute1.Velocity		:= PackTags.Command.Parameter[1].Value;
		stAxis.PTP.MoveAbsolute1.Position		:= (AxisMain.NcToPlc.ActPos + fConveyorLenght); 
		IF stAxis.PTP.MoveAbsolute1.Done THEN
			stAxis.PTP.MoveAbsolute1.Execute	:= FALSE;
			M_StateComplete();
		END_IF
										
	ePMLUnitMode_Service:		
		M_StateComplete();
END_CASE
END_METHOD

{attribute 'object_name' := 'M_Undefined'}
METHOD M_Undefined
bUndefinedDone	:= TRUE;
END_METHOD

END_FUNCTION_BLOCK

// ---- POUs/General/FB_AxisGeneral.TcPOU
//Functionblock for general axisbehavior
FUNCTION_BLOCK FB_AxisGeneral EXTENDS FB_Generic
VAR_IN_OUT
	Axis					: AXIS_REF;		//Axis reference
END_VAR
VAR_INPUT
	fConveyorLenght			: LREAL;		//Half Lenght of the Belt
	fConveyorVelo			: LREAL;		//Velocity from the Belt
	bMoveFw					: BOOL;			//Button for Manual Movement
END_VAR
VAR_OUTPUT
	bResettingDone			: BOOL;			//TRUE if Resetting is finished
END_VAR
VAR	
	stAxis					: ST_AxFunctions;		//Struct with motionfunctions
	iStateClearing			: INT;			//State variable for Clearing
	iStateResetting			: INT;			//State variable for Resetting
END_VAR

IF NOT (fbStateMachine.eState = ePMLState_Clearing) THEN
	iStateClearing	:= 0;
END_IF
IF NOT (fbStateMachine.eState = ePMLState_Resetting) THEN
	iStateResetting	:= 0; 
END_IF

this^.M_Reset();

//Call FB_Generic
SUPER^();

//Call the Motionfunctions from the ST_Axis
stAxis.Admin.Power(			Axis	:= Axis);
stAxis.Admin.Reset(			Axis	:= Axis);
stAxis.PTP.MoveAbsolute1(	Axis	:= Axis);
stAxis.PTP.MoveAbsolute2(	Axis	:= Axis);
stAxis.PTP.MoveVelocitiy(	Axis	:= Axis);
stAxis.PTP.Stop(			Axis	:= Axis);
stAxis.PTP.Halt(			Axis	:= Axis);

//Call the Axis, read NC parameters
Axis.ReadStatus();

{attribute 'object_name' := 'M_Aborting'}
METHOD M_Aborting
CASE fbUnitModeManager.eModeStatus OF
	ePMLProtUnitMode_Production, ePMLProtUnitMode_Manual:	

		bResettingDone			:= FALSE;
		iStateClearing		:= 0;
		
		IF NOT stAxis.PTP.Stop.Done AND stAxis.Admin.Power.Status THEN
			//Stop the axis
			stAxis.PTP.Stop.Deceleration		:= 0;
			stAxis.PTP.Stop.Execute				:= TRUE;
			stAxis.PTP.Stop.Jerk				:= 0;
			//take away the executes from MoveVelocity and MoveAbsolute
			 stAxis.PTP.MoveAbsolute1.Execute	:= FALSE;
			 stAxis.PTP.MoveAbsolute2.Execute	:= FALSE;
			 stAxis.PTP.MoveVelocitiy.Execute	:= FALSE;
		END_IF
		
		IF stAxis.PTP.Stop.Done THEN
			stAxis.PTP.Stop.Execute				:= FALSE;
			//Take away the SW-enalbe, so the user can move the belt with his hands  
			stAxis.Admin.Power.Enable			:= FALSE;
			stAxis.Admin.Power.Enable_Negative	:= FALSE;
			stAxis.Admin.Power.Enable_Positive	:= FALSE;
		END_IF
		
		IF NOT stAxis.Admin.Power.Status THEN
			M_StateComplete();
		END_IF
			
	ePMLProtUnitMode_Maintenance, ePMLUnitMode_Service:	
		M_StateComplete();
END_CASE
END_METHOD

{attribute 'object_name' := 'M_Clearing'}
METHOD M_Clearing
CASE fbUnitModeManager.eModeStatus OF
	ePMLProtUnitMode_Production, ePMLProtUnitMode_Manual:
		CASE iStateClearing OF 
			0:
				//Reset the Axis
				stAxis.Admin.Reset.Execute				:= TRUE;
				IF stAxis.Admin.Reset.Done  THEN
					stAxis.Admin.Reset.Execute			:= FALSE;
					iStateClearing								:= 1;
				END_IF
				IF stAxis.Admin.Reset.Error THEN
					iStateClearing								:= 0;
				END_IF
			1:	
				//Get the SW-Enable for the Axis
				stAxis.Admin.Power.BufferMode			:= MC_Aborting;
				stAxis.Admin.Power.Enable				:= TRUE;
				stAxis.Admin.Power.Enable_Negative		:= TRUE;
				stAxis.Admin.Power.Enable_Positive		:= TRUE;
				stAxis.Admin.Power.Override				:= 100.0;
				IF stAxis.Admin.Power.Status THEN
					M_StateComplete();
				END_IF
			END_CASE
			
	ePMLProtUnitMode_Maintenance, ePMLUnitMode_Service:
		M_StateComplete();
END_CASE
END_METHOD

{attribute 'object_name' := 'M_Completing'}
METHOD M_Completing
CASE fbUnitModeManager.eModeStatus OF 
	ePMLProtUnitMode_Production:			//Production, Mantainance, Manual	
		//disable the MC_MoveVeolocity
		stAxis.PTP.MoveVelocitiy.Execute	:= FALSE;
		stAxis.PTP.MoveAbsolute1.Execute	:= FALSE;
		stAxis.PTP.MoveAbsolute2.Execute	:= FALSE;
		IF PackTags.Status.StateCurrent = ePMLState_Completing THEN
			M_StateComplete();
		END_IF	
END_CASE
END_METHOD

{attribute 'object_name' := 'M_Execute'}
METHOD M_Execute
CASE fbUnitModeManager.eModeStatus OF		
	ePMLProtUnitMode_Production:
			
	ePMLProtUnitMode_Maintenance:		//Mantainancemode
		stAxis.PTP.Stop.Deceleration				:= 0;
		stAxis.PTP.Stop.Execute						:= TRUE;
		stAxis.PTP.Stop.Jerk						:= 0;
	
	ePMLProtUnitMode_Manual:		//Manualmode		
		IF bMoveFw THEN
			stAxis.PTP.Halt.Execute						:= FALSE;
			stAxis.PTP.MoveVelocitiy.Acceleration		:= 0;
			stAxis.PTP.MoveVelocitiy.BufferMode			:= MC_Aborting;
			stAxis.PTP.MoveVelocitiy.Deceleration		:= 0;
			stAxis.PTP.MoveVelocitiy.Direction			:= MC_Positive_Direction;
			stAxis.PTP.MoveVelocitiy.Execute			:= TRUE;
			stAxis.PTP.MoveVelocitiy.Jerk				:= 0;
			stAxis.PTP.MoveVelocitiy.Velocity			:= fConveyorVelo;
		ELSE
			stAxis.PTP.MoveVelocitiy.Execute			:= FALSE;
			stAxis.PTP.Halt.BufferMode					:= MC_Aborting;
			stAxis.PTP.Halt.Deceleration				:= 0;
			stAxis.PTP.Halt.Execute						:= TRUE;
			stAxis.PTP.Halt.Jerk						:= 0;
		END_IF

	ePMLUnitMode_Service:		//UserMode
			//Not defined
END_CASE
END_METHOD

{attribute 'object_name' := 'M_Idle'}
METHOD M_Idle
iStateResetting	:= 0;
END_METHOD

METHOD M_Reset
VAR_INPUT
END_VAR
IF stChangeIntoProduction.bYesReset THEN
	bMoveFw				:= FALSE;
	iStateClearing		:= 0;
	iStateResetting		:= 0;
END_IF
END_METHOD

{attribute 'object_name' := 'M_Resetting'}
METHOD M_Resetting
CASE fbUnitModeManager.eModeStatus OF
	ePMLProtUnitMode_Production:		
	
	ePMLProtUnitMode_Maintenance:

	ePMLProtUnitMode_Manual:		
		IF stAxis.Admin.Power.Status THEN
			iStateClearing		:= 0;
			M_StateComplete();
		ELSE
			stAxis.Admin.Power.BufferMode			:= MC_Aborting;
			stAxis.Admin.Power.Enable				:= TRUE;
			stAxis.Admin.Power.Enable_Negative		:= TRUE;
			stAxis.Admin.Power.Enable_Positive		:= TRUE;
			stAxis.Admin.Power.Override				:= 100.0;
		END_IF
		
	ePMLUnitMode_Service:				//Usermode
		//not defined	

END_CASE
END_METHOD

{attribute 'object_name' := 'M_Starting'}
METHOD M_Starting
CASE fbUnitModeManager.eModeStatus OF
	ePMLProtUnitMode_Production, ePMLProtUnitMode_Manual:		
		bResettingDone			:= FALSE;
		stAxis.PTP.Halt.Execute					:= FALSE;
		stAxis.PTP.MoveAbsolute1.Execute		:= FALSE;
		stAxis.PTP.MoveAbsolute2.Execute		:= FALSE;
		stAxis.PTP.MoveVelocitiy.Execute		:= FALSE;
		stAxis.PTP.Stop.Execute					:= FALSE;
		iStateResetting									:= 0;
		SUPER^.M_Starting();
					
	ePMLProtUnitMode_Maintenance, ePMLUnitMode_Service:			
		SUPER^.M_Starting();
END_CASE
END_METHOD

{attribute 'object_name' := 'M_Stopped'}
METHOD M_Stopped
iStateResetting	:= 0;
END_METHOD

{attribute 'object_name' := 'M_Stopping'}
METHOD M_Stopping
CASE fbUnitModeManager.eModeStatus OF
	ePMLProtUnitMode_Production, ePMLProtUnitMode_Manual:	
		bResettingDone			:= FALSE;
		
		IF NOT stAxis.PTP.Stop.Done AND stAxis.Admin.Power.Status THEN
			//Stop the Axis
			stAxis.PTP.Stop.Deceleration		:= 0;
			stAxis.PTP.Stop.Execute				:= TRUE;
			stAxis.PTP.Stop.Jerk				:= 0;
			//take away the Executes from MoveVelocity and Move absolte
			 stAxis.PTP.MoveAbsolute1.Execute	:= FALSE;
			 stAxis.PTP.MoveVelocitiy.Execute	:= FALSE;
		END_IF
		
		IF stAxis.PTP.Stop.Done THEN
			stAxis.PTP.Stop.Execute				:= FALSE;
			//Take away the SW-enalbe, so the user can move the belt with his hands  
			stAxis.Admin.Power.Enable			:= FALSE;
			stAxis.Admin.Power.Enable_Negative	:= FALSE;
			stAxis.Admin.Power.Enable_Positive	:= FALSE;
		END_IF
		
		IF NOT stAxis.Admin.Power.Status THEN
			M_StateComplete();
		END_IF
			
	ePMLProtUnitMode_Maintenance, ePMLUnitMode_Service:
		M_StateComplete();
END_CASE
END_METHOD

{attribute 'object_name' := 'M_Unholding'}
METHOD M_Unholding
CASE fbUnitModeManager.eModeStatus OF
	ePMLProtUnitMode_Production:			//Production
		IF  PackTags.Status.StateCurrent = ePMLState_Unholding THEN
			M_StateComplete();
		END_IF
				
	ePMLProtUnitMode_Maintenance, ePMLUnitMode_Service:			//Mantainance & UserMode
		M_StateComplete();
END_CASE
END_METHOD

{attribute 'object_name' := 'M_Unsuspending'}
METHOD M_Unsuspending
CASE fbUnitModeManager.eModeStatus OF
	ePMLProtUnitMode_Production:			//Production
		IF PackTags.Status.StateCurrent = ePMLState_Unsuspending THEN
			M_StateComplete();
		END_IF
					
	ePMLUnitMode_Service:			//Usermode
		M_StateComplete();	
END_CASE
END_METHOD

END_FUNCTION_BLOCK

// ---- POUs/Units/Seperation/FB_Seperation.TcPOU
FUNCTION_BLOCK FB_Seperation EXTENDS FB_Generic
VAR_INPUT
	bMoveBarrierCylinder				: BOOL;				//Button to move Barriercylinder
	bMoveClambCylinder					: BOOL;				//Button to move Clamber
END_VAR
VAR_OUTPUT
	bMoveToWorkBarrierHW				: BOOL;				//Barrier moves to workposition, utput for FB_Visu
	bMoveToWorkClambHW					: BOOL;				//Clamber moves to workposition, utput for FB_Visu
END_VAR
VAR	
	fbCylinderClamb						: FB_Cylinder;		//Subunit1
	fbCylinderBarrier					: FB_Cylinder;		//Subunit2

	nStateExecute						: INT;				//State for processing the Seperation
	fbTimerSeperation					: TON;				//Timer for waiting, till the Box is on mainbelt
	
	bSensorBarrier	AT%I*				: BOOL;				//Sensor to detct a box at the barriercylinder, link to PlcOutput fbVisu.bBarrierSensor
	
	//Counting Packtags
	fbTrigger							:F_TRIG;			//Trigger for counting the seperated boxes

END_VAR

SUPER^();

//Outreach the Variables in the FB_Machine
bMoveToWorkBarrierHW	:= fbCylinderBarrier.bMoveToWorkHW;
bMoveToWorkClambHW		:= fbCylinderClamb.bMoveToWorkHW;

//counting products and calculate the productionvelocity
fbTrigger(CLK:= fbCylinderBarrier.bAtWorkPos);
IF fbTrigger.Q AND fbUnitModeManager.eModeStatus = 1
  AND (fbStateMachine.eState =  ePMLState_Execute OR fbStateMachine.eState = ePMLState_Suspending OR
       fbStateMachine.eState = ePMLState_Holding OR fbStateMachine.eState = ePMLState_Resetting ) THEN	
	PackTags.Admin.ProdProcessedCount[2].Count		:=  PackTags.Admin.ProdProcessedCount[2].Count +1;
END_IF

THIS^.M_Reset();
fbCylinderBarrier();
fbCylinderClamb();
fbTimerSeperation();

{attribute 'object_name' := 'M_Aborting'}
METHOD M_Aborting
CASE fbUnitModeManager.eModeStatus OF	
	ePMLProtUnitMode_Production, ePMLProtUnitMode_Manual:		
		IF fbCylinderBarrier.bAtBasePos THEN
			fbCylinderBarrier.bMoveToWork	:= FALSE;
		END_IF
		IF fbCylinderClamb.bAtBasePos THEN
			fbCylinderClamb.bMoveToWork		:= FALSE;
		END_IF
		fbTimerSeperation.IN	:= FALSE;
		M_StateComplete();
			
	ePMLProtUnitMode_Maintenance, ePMLUnitMode_Service:
		M_StateComplete();
END_CASE
END_METHOD

{attribute 'object_name' := 'M_Completing'}
METHOD M_Completing
CASE fbUnitModeManager.eModeStatus OF
	ePMLProtUnitMode_Production:
		//Waiting till all units are in Completing
		IF PackTags.Status.StateCurrent = ePMLState_Completing THEN
			M_StateComplete();
		END_IF
END_CASE
END_METHOD

{attribute 'object_name' := 'M_Execute'}
METHOD M_Execute

VAR

END_VAR
CASE fbUnitModeManager.eModeStatus OF
	ePMLProtUnitMode_Production:		//Mode Production
		//Processing automatic Seperation
		CASE nStateExecute OF
			0:
				IF	PackTags.Admin.ProdProcessedCount[2].Count >= REAL_TO_DINT( PackTags.Command.Parameter[2].Value) AND  PackTags.Admin.ProdProcessedCount[1].Count = REAL_TO_DINT(PackTags.Command.Parameter[2].Value)AND
					fbCylinderBarrier.bAtBasePos AND  AxisMain.Status.NotMoving AND AxisPlastic.Status.NotMoving AND AxisMetal.Status.NotMoving AND
					PackTags.Status.StateCurrent = ePMLState_Execute THEN
						M_StateComplete();
				ELSIF PackTags.Admin.ProdProcessedCount[2].Count >= REAL_TO_DINT( PackTags.Command.Parameter[2].Value) AND fbCylinderBarrier.bAtBasePos AND fbCylinderClamb.bAtBasePos THEN
						nStateExecute			:= 0;
				ELSE
						nStateExecute			:= 1;
				END_IF
				
			1:	
				fbCylinderClamb.bMoveToWork		:=	FALSE; 
				fbCylinderBarrier.bMoveToWork	:=	TRUE;
				IF 	 fbCylinderBarrier.bAtWorkPos THEN
					nStateExecute				:= 2;
				END_IF
			2:
				fbTimerSeperation.IN	:= TRUE; 
				fbTimerSeperation.PT	:= T#4S;
				IF fbTimerSeperation.Q THEN
					fbTimerSeperation.IN			:= FALSE;
					nStateExecute				:= 3;
				END_IF
				
			3:
				fbCylinderBarrier.bMoveToWork	:=	FALSE;
				IF fbCylinderBarrier.bAtBasePos THEN
					nStateExecute				:= 4;
				END_IF
				
			4:
				fbCylinderClamb.bMoveToWork		:=	TRUE;
				IF fbCylinderClamb.bAtWorkPos AND bSensorBarrier THEN
					nStateExecute				:= 5;
				END_IF
			5:
				fbCylinderClamb.bMoveToWork		:=	FALSE;
				IF fbCylinderClamb.bAtBasePos AND fbCylinderBarrier.bAtBasePos THEN
					nStateExecute				:= 0;
				END_IF
		END_CASE

	ePMLProtUnitMode_Maintenance, ePMLUnitMode_Service:		
		//
		
	ePMLProtUnitMode_Manual:		//Manaul
		//React on Visubuttons		
		IF  bMoveBarrierCylinder THEN
			fbCylinderBarrier.bMoveToWork	:=	TRUE;
		ELSE
			fbCylinderBarrier.bMoveToWork	:=	FALSE;
		END_IF
		IF bMoveClambCylinder	THEN
			fbCylinderClamb.bMoveToWork		:=	TRUE;
		ELSE
			fbCylinderClamb.bMoveToWork		:=	FALSE;
		END_IF
END_CASE
END_METHOD

{attribute 'object_name' := 'M_Holding'}
METHOD M_Holding
CASE fbUnitModeManager.eModeStatus OF
	ePMLProtUnitMode_Production:		//Mode Production
		//Finisch the actual seperationstep	
		CASE nStateExecute OF
			0:
				M_StateComplete();	
			1:	
				fbCylinderClamb.bMoveToWork		:=	FALSE; 
				fbCylinderBarrier.bMoveToWork	:=	TRUE;
				IF 	 fbCylinderBarrier.bAtWorkPos THEN
					nStateExecute				:= 2;
				END_IF
			2:
				fbTimerSeperation.IN	:= TRUE; 
				fbTimerSeperation.PT	:= T#4S;
				IF fbTimerSeperation.Q THEN
					fbTimerSeperation.IN			:= FALSE;
					nStateExecute				:= 3;
				END_IF
				
			3:
				fbCylinderBarrier.bMoveToWork	:=	FALSE;
				IF fbCylinderBarrier.bAtBasePos THEN
					nStateExecute				:= 4;
				END_IF
					
			4:
				fbCylinderClamb.bMoveToWork		:=	TRUE;
				IF fbCylinderClamb.bAtWorkPos AND bSensorBarrier THEN
					nStateExecute				:= 5;
				END_IF
			5:
				fbCylinderClamb.bMoveToWork		:=	FALSE;
				IF fbCylinderClamb.bAtBasePos AND fbCylinderBarrier.bAtBasePos THEN
					nStateExecute				:= 5;
					M_StateComplete();
				END_IF
		END_CASE

	ePMLProtUnitMode_Maintenance:
		M_StateComplete();
END_CASE
END_METHOD

METHOD M_Reset
VAR_INPUT
END_VAR
//Take away all commands
IF stChangeIntoProduction.bYesReset THEN
	nStateExecute					:= 0;
	fbTimerSeperation.IN			:= FALSE;
	fbCylinderBarrier.bMoveToWork	:= FALSE;
	fbCylinderClamb.bMoveToWork		:= FALSE;
END_IF
END_METHOD

{attribute 'object_name' := 'M_Resetting'}
METHOD M_Resetting
CASE fbUnitModeManager.eModeStatus OF
	ePMLProtUnitMode_Production:		//Production, Mantainance, Manual	
		IF nStateExecute = 0 AND fbCylinderBarrier.bAtBasePos AND fbCylinderClamb.bAtBasePos AND bSensorBarrier THEN
			M_StateComplete();
		ELSIF AxisMain.Status.Moving THEN
			//Finisch the actual seperationstep	
			CASE nStateExecute OF
			0:
				M_StateComplete();									
				fbCylinderClamb.bMoveToWork		:=	FALSE;
				fbCylinderBarrier.bMoveToWork	:=	FALSE;			
			1:	
				fbCylinderClamb.bMoveToWork		:=	FALSE; 
				fbCylinderBarrier.bMoveToWork	:=	TRUE;
				IF 	 fbCylinderBarrier.bAtWorkPos THEN
					nStateExecute				:= 2;
				END_IF
			2:
				fbTimerSeperation.IN	:= TRUE; 
				fbTimerSeperation.PT	:= T#4S;
				IF fbTimerSeperation.Q THEN
					fbTimerSeperation.IN			:= FALSE;
					nStateExecute				:= 3;
				END_IF
					
			3:
				fbCylinderBarrier.bMoveToWork	:=	FALSE;
				IF fbCylinderBarrier.bAtBasePos THEN
					nStateExecute				:= 4;
				END_IF
						
			4:
				fbCylinderClamb.bMoveToWork		:=	TRUE;
				IF fbCylinderClamb.bAtWorkPos AND bSensorBarrier THEN
					nStateExecute				:= 5;
				END_IF
			5:
				fbCylinderClamb.bMoveToWork		:=	FALSE;
				IF fbCylinderClamb.bAtBasePos AND fbCylinderBarrier.bAtBasePos THEN
					nStateExecute				:= 0;
				END_IF
			END_CASE
		END_IF
	
	ePMLProtUnitMode_Maintenance, ePMLProtUnitMode_Manual, ePMLUnitMode_Service:
		M_StateComplete();
END_CASE
END_METHOD

{attribute 'object_name' := 'M_Starting'}
METHOD M_Starting
CASE fbUnitModeManager.eModeStatus OF
	ePMLProtUnitMode_Production:		//Production, Mantainance, Manual
		//Resetting all Commands and Values
		fbTimerSeperation.IN			:= FALSE;
		nStateExecute					:= 0;
		fbCylinderBarrier.bMoveToWork	:= FALSE;
		fbCylinderClamb.bMoveToWork		:= FALSE;
		IF fbCylinderBarrier.bAtBasePos AND fbCylinderClamb.bAtBasePos THEN
			SUPER^.M_Starting();
		END_IF

	ePMLProtUnitMode_Maintenance, ePMLProtUnitMode_Manual, ePMLUnitMode_Service:
		M_StateComplete();
END_CASE
END_METHOD

{attribute 'object_name' := 'M_Stopping'}
METHOD M_Stopping
CASE fbUnitModeManager.eModeStatus OF
	ePMLProtUnitMode_Production, ePMLProtUnitMode_Manual:			
		IF fbCylinderBarrier.bAtBasePos THEN
			fbCylinderBarrier.bMoveToWork	:= FALSE;
		END_IF
		IF fbCylinderClamb.bAtBasePos THEN
			fbCylinderClamb.bMoveToWork		:= FALSE;
		END_IF
		fbTimerSeperation.IN	:= FALSE;
		M_StateComplete();

	ePMLProtUnitMode_Maintenance, ePMLUnitMode_Service:
		M_StateComplete();	
			//not defined
END_CASE
END_METHOD

{attribute 'object_name' := 'M_Suspending'}
METHOD M_Suspending
CASE fbUnitModeManager.eModeStatus OF
	ePMLProtUnitMode_Production:		//Mode Production
		//Finisch the actual seperationstep	
		CASE nStateExecute OF
			0:
				M_StateComplete();	
			1:	
				fbCylinderClamb.bMoveToWork		:=	FALSE; 
				fbCylinderBarrier.bMoveToWork	:=	TRUE;
				IF 	 fbCylinderBarrier.bAtWorkPos THEN
					nStateExecute				:= 2;
				END_IF
			2:
				fbTimerSeperation.IN	:= TRUE; 
				fbTimerSeperation.PT	:= T#4S;
				IF fbTimerSeperation.Q THEN
					fbTimerSeperation.IN			:= FALSE;
					nStateExecute				:= 3;
				END_IF
			3:
				fbCylinderBarrier.bMoveToWork	:=	FALSE;
				IF fbCylinderBarrier.bAtBasePos THEN
					nStateExecute				:= 4;
				END_IF
					
			4:
				fbCylinderClamb.bMoveToWork		:=	TRUE;
				IF fbCylinderClamb.bAtWorkPos AND bSensorBarrier THEN
					nStateExecute				:= 5;
				END_IF
			5:
				fbCylinderClamb.bMoveToWork		:=	FALSE;
				IF fbCylinderClamb.bAtBasePos AND fbCylinderBarrier.bAtBasePos THEN
					nStateExecute				:= 5;
					M_StateComplete();
				END_IF
		END_CASE

	ePMLUnitMode_Service:
		M_StateComplete();
END_CASE
END_METHOD

{attribute 'object_name' := 'M_Undefined'}
METHOD M_Undefined
fbCylinderBarrier.bMoveToWork	:= FALSE;
fbCylinderClamb.bMoveToWork		:= FALSE;
bUndefinedDone					:= TRUE;
END_METHOD

{attribute 'object_name' := 'M_Unholding'}
METHOD M_Unholding
CASE fbUnitModeManager.eModeStatus OF
	ePMLProtUnitMode_Production:	//Production, Mantainance, Manual
		IF fbCylinderBarrier.bAtBasePos AND fbCylinderClamb.bAtBasePos AND PackTags.Status.StateCurrent = ePMLState_Unholding THEN
			M_StateComplete();
			nStateExecute		:= 0;
			fbTimerSeperation.IN	:= FALSE;
		END_IF
			
	ePMLProtUnitMode_Maintenance, ePMLUnitMode_Service:	
		M_StateComplete();
END_CASE
END_METHOD

{attribute 'object_name' := 'M_Unsuspending'}
METHOD M_Unsuspending
CASE fbUnitModeManager.eModeStatus OF
	ePMLProtUnitMode_Production:	//Production, Mantainance, Manual
		IF fbCylinderBarrier.bAtBasePos AND fbCylinderClamb.bAtBasePos AND PackTags.Status.StateCurrent = ePMLState_Unsuspending THEN
			M_StateComplete();
			nStateExecute		:= 0;
			fbTimerSeperation.IN	:= FALSE;
		END_IF	

	ePMLUnitMode_Service:			
		M_StateComplete();
END_CASE
END_METHOD

END_FUNCTION_BLOCK

// ---- POUs/General/FB_Cylinder.TcPOU
FUNCTION_BLOCK FB_Cylinder 
VAR_INPUT
	bMoveToWork					: BOOL;		//Command, that cylinder move to work position
END_VAR
VAR_OUTPUT
	bMoveToWorkHW	AT%Q*		: BOOL;		//HW-Signal output, cylinder move to workposition
	bAtBasePos		AT%I*		: BOOL;		//HW-Signal input, cylinder in baseposition
	bAtWorkPos		AT%I*		: BOOL;		//HW-Signal input, cylinder in workposition
END_VAR

IF bMoveToWork THEN
	bMoveToWorkHW	:= TRUE;
ELSE
	bMoveToWorkHW	:= FALSE;
END_IF

END_FUNCTION_BLOCK

// ---- POUs/Units/Ejection/FB_Ejector.TcPOU
FUNCTION_BLOCK FB_Ejector EXTENDS FB_Generic
VAR_IN_OUT
	Axis							: AXIS_REF;		//Axis reference
END_VAR
VAR_INPUT
	bMoveBeltFw						: BOOL;			//Variable to move Belt forward, link to FB_Visu
	bMoveCylinder					: BOOL;			//Variable to move cylinder to workposition, link to FB_Visu
	bSensorEjection		AT%I*		: BOOL;			//HW-Signal input, detection of boxes, link to TC3_PackML_Simu
END_VAR
VAR_OUTPUT
	bMoveToWork						: BOOL;			//Varaible to outreach the actual command for the cylindermovement in the FB_Machine -> FB_Visu
	bResetDone						: BOOL;			//TRUE, if subunits have succesfull resetting. Link to GVL: bMetalEjectionResetDone and bPlasticEjectionResetDone
	nCounterProduct					: DINT :=0;		//Varible for counting only finished metal- and plasticboxes. Link to PackTags.Admin.ProdProcessedCount[3] AND PackTags.Admin.ProdProcessedCount[4]
	
	eModeSensor						: DINT;			//Mode from the subunit sensor
	eStateSesnor					: E_PMLState;	//State from the subunit sensor
	eModeAxis						: DINT;			//Mode from the subunit axis
	eStateAxis						: E_PMLState;	//State from the subunit axis
END_VAR
VAR
	fbCylinderEjection				: FB_Cylinder;	//Cylinder to eject boxes
	
	fbSensorEjection				: FB_Sensor;	//Sensor to detect boxes, with delaytime and breakfunction
	
	R_Trigger						: R_TRIG;		//Trigger for counting finished Boxes
	fTrigger						: F_TRIG;		//Trigger for setting nCounterProduct to 0
	

	fbAxisEjection					: FB_AxixEjection;						//Axis to dispatch boxes
	stSubUnitInfo					: ARRAY [1..2] OF ST_PMLSubUnitInfo;	//Informations about the subunits
END_VAR

//Call FB_Cylinder
fbCylinderEjection();

//Call FB_AxixEjection
fbAxisEjection(		
	Axis				:= Axis,
	eModeCommand		:= eModeCommand,
	eCommand			:= eCommand,
	fConveyorLenght		:= 300.0,
	bStartBelt			:= fbCylinderEjection.bAtWorkPos,
	fConveyorVelo		:= PackTags.Command.Parameter[3].Value,
	bMoveFw 			:= bMoveBeltFw,
	eMode				=>,
	eState				=> stSubUnitInfo[1].eState,
	bResettingDone 		=> bResetDone);	
stSubUnitInfo[1].Active			:= TRUE;
eModeAxis						:= fbAxisEjection.eMode;
eStateAxis						:= fbAxisEjection.eState;

//Call FB_Sensor
fbSensorEjection(	
	Axis			:= Axis,
	eModeCommand	:= eModeCommand,
	eCommand		:= eCommand, 
	tDelayTime		:= T#2S950MS,
	eMode 			=> ,
	eState			=> stSubUnitInfo[2].eState);

stSubUnitInfo[2].Active		:= TRUE;
eModeSensor					:= fbSensorEjection.eMode;
eStateSesnor				:= fbSensorEjection.eState;

//The fbStateMachine from FB_Ejector gets the Information about the states and activity from the subunits
fbStateMachine.stSubUnitInfoRef.ArraySize		:= SIZEOF(stSubUnitInfo);
fbStateMachine.stSubUnitInfoRef.NoOfSubUnits	:= 2;
fbStateMachine.stSubUnitInfoRef.pArray			:= ADR(stSubUnitInfo);

//Outreach the actual movementcommand for the cylinder in the FB_Machine -> FB_Visu
bMoveToWork	:= fbCylinderEjection.bMoveToWorkHW;

//Counting all finished plastic- and metalboxes
R_Trigger(CLK:= fbCylinderEjection.bAtWorkPos );
IF	R_Trigger.Q	AND fbUnitModeManager.eModeStatus = 1 THEN
		PackTags.Admin.ProdProcessedCount[1].AccCount	:= PackTags.Admin.ProdProcessedCount[1].AccCount +1;
		PackTags.Admin.ProdProcessedCount[1].Count		:= PackTags.Admin.ProdProcessedCount[1].Count	 +1;
		nCounterProduct									:= nCounterProduct +1;
END_IF

//Reset the counter when production has finished
fTrigger(CLK:= (fbStateMachine.eState = ePMLState_Complete) );
IF fTrigger.Q OR stChangeIntoProduction.bYesReset THEN
		nCounterProduct	:= 0;
END_IF

//Call the reset method from FB_Ejector
this^.M_Reset();

//Call FB_Generic
SUPER^();

{attribute 'object_name' := 'M_Aborting'}
METHOD M_Aborting
CASE fbUnitModeManager.eModeStatus OF
	ePMLProtUnitMode_Production, ePMLProtUnitMode_Manual:	//Manual, Mantainance, Manual
		//finish the actaul movement from the cylinder
		IF fbCylinderEjection.bAtBasePos OR fbCylinderEjection.bAtWorkPos THEN
			M_StateComplete();
		END_IF
		
	ePMLProtUnitMode_Maintenance, ePMLUnitMode_Service:
		M_StateComplete();
END_CASE
END_METHOD

{attribute 'object_name' := 'M_Completing'}
METHOD M_Completing
CASE fbUnitModeManager.eModeStatus OF
	ePMLProtUnitMode_Production:
		//Waiting till all subunits are in the state completing
		IF PackTags.Status.StateCurrent  = ePMLState_Completing THEN
			M_StateComplete();
		END_IF
END_CASE
END_METHOD

{attribute 'object_name' := 'M_Execute'}
METHOD M_Execute
CASE fbUnitModeManager.eModeStatus OF
	ePMLProtUnitMode_Production:		//Production
		//Ejection from Metalboxes
		fbSensorEjection.bInput			:= bSensorEjection;
		
		IF fbSensorEjection.bOutput  THEN
			fbCylinderEjection.bMoveToWork			:= TRUE;
		END_IF
		
		IF fbCylinderEjection.bAtWorkPos THEN
			fbCylinderEjection.bMoveToWork		:= FALSE;
		END_IF
		
		//Production of command products is finished
		IF REAL_TO_DINT(PackTags.Command.Parameter[2].Value) <=  PackTags.Admin.ProdProcessedCount[1].Count AND
			AxisMain.Status.NotMoving AND AxisPlastic.Status.NotMoving AND AxisMetal.Status.NotMoving AND fbCylinderEjection.bAtBasePos AND
			PackTags.Status.StateCurrent = ePMLState_Execute THEN
			M_StateComplete();
		END_IF
		
	ePMLProtUnitMode_Maintenance, ePMLUnitMode_Service:		
		//
		
	ePMLProtUnitMode_Manual:		//Manual
		IF bMoveCylinder THEN
			fbCylinderEjection.bMoveToWork		:= TRUE;
		ELSE
			fbCylinderEjection.bMoveToWork		:= FALSE;
		END_IF
END_CASE
END_METHOD

{attribute 'object_name' := 'M_Holding'}
METHOD M_Holding
CASE fbUnitModeManager.eModeStatus OF
	ePMLProtUnitMode_Production:		//Production	
		//Ejection from boxes
		fbSensorEjection.bInput					:= bSensorEjection;

		IF fbSensorEjection.bOutput  THEN
			fbCylinderEjection.bMoveToWork		:= TRUE;
		END_IF
		IF fbCylinderEjection.bAtWorkPos THEN
			fbCylinderEjection.bMoveToWork		:= FALSE;
			
		END_IF

		//Conveyor stops working
		IF AxisMain.Status.NotMoving AND AxisPlastic.Status.NotMoving AND AxisMetal.Status.NotMoving AND fbCylinderEjection.bAtBasePos THEN
			fbCylinderEjection.bMoveToWork		:= FALSE;
			M_StateComplete();
		END_IF

	ePMLProtUnitMode_Maintenance:
		M_StateComplete();
END_CASE
END_METHOD

METHOD M_Reset
VAR_INPUT
END_VAR
IF stChangeIntoProduction.bYesReset THEN
	fbCylinderEjection.bMoveToWork := FALSE;
END_IF
END_METHOD

{attribute 'object_name' := 'M_Resetting'}
METHOD M_Resetting
CASE fbUnitModeManager.eModeStatus OF	
	ePMLProtUnitMode_Production:		//Production, Mantainance, Manaul Mode
		fbSensorEjection.bInput			:= bSensorEjection;
		IF bSensorEjection THEN
			fbSensorEjection.tDelayTime	:= T#3S;
		END_IF

		IF fbSensorEjection.bOutput  THEN
			fbCylinderEjection.bMoveToWork			:= TRUE;
		END_IF
		IF fbCylinderEjection.bAtWorkPos THEN
			fbCylinderEjection.bMoveToWork		:= FALSE;
		END_IF

		
		
		IF bAxisMainResetDone AND  fbCylinderEjection.bAtBasePos THEN
			M_StateComplete();
		END_IF

	ePMLProtUnitMode_Maintenance, ePMLProtUnitMode_Manual, ePMLUnitMode_Service:
		M_StateComplete();
END_CASE
END_METHOD

{attribute 'object_name' := 'M_Stopping'}
METHOD M_Stopping
CASE fbUnitModeManager.eModeStatus OF
	ePMLProtUnitMode_Production, ePMLProtUnitMode_Manual:
		IF fbCylinderEjection.bAtBasePos OR fbCylinderEjection.bAtWorkPos THEN
			M_StateComplete();
		END_IF

	ePMLProtUnitMode_Maintenance, ePMLUnitMode_Service:
		M_StateComplete();
END_CASE
END_METHOD

{attribute 'object_name' := 'M_Suspending'}
METHOD M_Suspending
CASE fbUnitModeManager.eModeStatus OF
	ePMLProtUnitMode_Production:		//Production	
		//Ejection from boxes
		fbSensorEjection.bInput			:= bSensorEjection;
		IF bSensorEjection THEN
			fbSensorEjection.tDelayTime	:= T#3S;
		END_IF

		IF fbSensorEjection.bOutput  THEN
			fbCylinderEjection.bMoveToWork			:= TRUE;
		END_IF
		IF fbCylinderEjection.bAtWorkPos THEN
			fbCylinderEjection.bMoveToWork		:= FALSE;
		END_IF
		
		//Conveyor stops working
		IF AxisMain.Status.NotMoving AND AxisPlastic.Status.NotMoving AND AxisMetal.Status.NotMoving AND fbCylinderEjection.bAtBasePos THEN
			fbCylinderEjection.bMoveToWork		:= FALSE;
			M_StateComplete();
		END_IF

	ePMLUnitMode_Service:
		M_StateComplete();
END_CASE
END_METHOD

{attribute 'object_name' := 'M_Undefined'}
METHOD M_Undefined
fbCylinderEjection.bMoveToWork		:= FALSE;
IF fbAxisejection.bUndefinedDone AND fbSensorEjection.bUndefinedDone  THEN
	bUndefinedDone					:= TRUE;
END_IF
END_METHOD

{attribute 'object_name' := 'M_Unholding'}
METHOD M_Unholding

CASE fbUnitModeManager.eModeStatus OF
	ePMLProtUnitMode_Production:
		IF PackTags.Status.StateCurrent = ePMLState_Unholding THEN
			M_StateComplete();
		END_IF

	ePMLProtUnitMode_Maintenance, ePMLUnitMode_Service:
		M_StateComplete();
END_CASE
END_METHOD

{attribute 'object_name' := 'M_Unsuspending'}
METHOD M_Unsuspending
//Waiting for subunits
IF PackTags.Status.StateCurrent = ePMLState_Unsuspending THEN
	M_StateComplete();
END_IF
END_METHOD

END_FUNCTION_BLOCK

// ---- POUs/Units/Ejection/FB_Sensor.TcPOU
FUNCTION_BLOCK FB_Sensor EXTENDS FB_Generic
VAR_IN_OUT
	Axis			: AXIS_REF;
END_VAR
VAR_INPUT
	tDelayTime		: TIME;			//delaytime
	bInput			: BOOL;			//HW-Signal from Sensor
END_VAR
VAR_OUTPUT
	bOutput			: BOOL;			//Output with delaytime
END_VAR
VAR
	fbTimer			: Ton_Break;	//Timer for delaytime witch breakfunction
	fbTriggerR		: R_Trig;		//Trigger to detect rising edge of HW-siganl
	nSensorState	: INT := 0;		//State variable for sensor - process to get siganl with delaytime
END_VAR

//Process to get siganl with delaytime
fbTriggerR(CLK := bInput);
CASE nSensorState OF
0:
	bOutput		:= FALSE;
	IF fbTriggerR.Q THEN
		nSensorState := 1;

	END_IF
		
1:
	fbTimer.IN	:= TRUE;
	IF fbTimer.Q THEN
		fbTimer.IN	:= FALSE;
		bOutput		:= TRUE;
		nSensorState:= 0;
	END_IF
END_CASE


//resetting Timer
IF stChangeIntoProduction.bYesReset THEN
	fbTimer.IN		:= FALSE;
	fbTimer.Halt	:= FALSE;
END_IF

//Resetting Timer 
IF PackTags.Status.UnitModeCurrent <> 1 THEN
	fbTimer.IN		:= FALSE;
	fbTimer.Halt	:= FALSE;
END_IF


fbTimer(PT	:= tDelayTime);


Super^();

{attribute 'object_name' := 'M_Aborting'}
METHOD M_Aborting
CASE fbUnitModeManager.eModeStatus OF
	ePMLProtUnitMode_Production:
		fbTimer.Halt := TRUE;
		M_StateComplete();

	ePMLProtUnitMode_Maintenance, ePMLProtUnitMode_Manual, ePMLUnitMode_Service:
		M_StateComplete();
END_CASE
END_METHOD

{attribute 'object_name' := 'M_Execute'}
METHOD M_Execute
CASE fbUnitModeManager.eModeStatus OF
	ePMLProtUnitMode_Production:		
		IF REAL_TO_DINT(PackTags.Command.Parameter[2].Value) <= PackTags.Admin.ProdProcessedCount[1].Count 
		  AND Axis.Status.NotMoving	
		  AND PackTags.Status.StateCurrent = ePMLState_Execute THEN
			M_StateComplete();
		END_IF
			
		IF  AxisMain.Status.Moving THEN
			fbTimer.Halt	:= FALSE;
		END_IF
	
	ePMLProtUnitMode_Maintenance, ePMLProtUnitMode_Manual, ePMLUnitMode_Service:
		//
END_CASE
END_METHOD

{attribute 'object_name' := 'M_Resetting'}
METHOD M_Resetting
CASE fbUnitModeManager.eModeStatus OF
	ePMLProtUnitMode_Production:
		IF AxisMain.Status.Moving THEN
			fbTimer.Halt	:= FALSE;
			M_StateComplete();
		END_IF
		
	ePMLProtUnitMode_Maintenance, ePMLProtUnitMode_Manual, ePMLUnitMode_Service:
		M_StateComplete();
END_CASE
END_METHOD

{attribute 'object_name' := 'M_Stopping'}
METHOD M_Stopping
CASE fbUnitModeManager.eModeStatus OF
	ePMLProtUnitMode_Production:
		fbTimer.Halt := TRUE;
		M_StateComplete();
		
	ePMLProtUnitMode_Maintenance, ePMLProtUnitMode_Manual, ePMLUnitMode_Service:
		M_StateComplete();
END_CASE
END_METHOD

{attribute 'object_name' := 'M_Undefined'}
METHOD M_Undefined
bUndefinedDone	:= TRUE;
END_METHOD

END_FUNCTION_BLOCK

// ---- POUs/General/Ton_Break.TcPOU
FUNCTION_BLOCK Ton_Break 
VAR_INPUT
	PT			: TIME;						//Time for Timer
	IN			: BOOL;						//Start timer
	Halt		: BOOL;						//halt timer
END_VAR
VAR_OUTPUT
	ET			: TIME;						//Outreach ET from Timer1
	Q			: BOOL;						//Outreach Q from Timer1
END_VAR
VAR
	Timer1		: Ton;						//Timer for delaytime
	PTintern	: TIME 	:= T#71582M47S295MS;//Max Range of Time

END_VAR

//checking if Halt is TRUE
IF Halt AND PTintern = T#71582M47S295MS THEN
	PTintern	:= Timer1.PT - Timer1.ET;
	Timer1.IN	:= FALSE;
ELSIF  PTintern < PT AND NOT Halt THEN
	Timer1.IN	:= IN;
	Timer1.PT	:= PTintern;
ELSIF NOT HALT THEN
	Timer1.IN	:= IN;
	Timer1.PT	:= PT;
END_IF

//Calling Timer
Timer1();
//Outreach Variables
Q	:= Timer1.Q;
ET	:= Timer1.ET;

//Settting PT on Max Value
IF  NOT IN  THEN
	PTintern	:= T#71582M47S295MS; 
END_IF

END_FUNCTION_BLOCK

// ---- POUs/Units/Ejection/FB_AxixEjection.TcPOU
FUNCTION_BLOCK FB_AxixEjection EXTENDS FB_AxisGeneral
VAR_INPUT
	bStartBelt	: BOOL;
END_VAR
VAR_OUTPUT
END_VAR
VAR
	TrigbStartbelt	: R_TRIG;
END_VAR

//Call the FB_Axis_General
SUPER^(Axis := Axis);

TrigbStartbelt(CLK:= bStartBelt);

{attribute 'object_name' := 'M_Completing'}
METHOD M_Completing
CASE fbUnitModeManager.eModeStatus OF 
	ePMLProtUnitMode_Production:			//Production
		//Stop the Axis
		stAxis.PTP.MoveVelocitiy.Execute	:= FALSE;
		stAxis.PTP.Stop.Deceleration		:= 500;
		stAxis.PTP.Stop.Execute				:= TRUE;
		stAxis.PTP.Stop.Jerk				:= 0;
		
		IF stAxis.PTP.Stop.Done AND PackTags.Status.StateCurrent = ePMLState_Completing THEN
			M_StateComplete();
		END_IF			
END_CASE
END_METHOD

{attribute 'object_name' := 'M_Execute'}
METHOD M_Execute
CASE fbUnitModeManager.eModeStatus OF
	ePMLProtUnitMode_Production:		
		//Use two MoveAbsolute functionblocks, to use the Buffermode MC_BlendingNext
		IF TrigbStartbelt.Q AND (stAxis.PTP.MoveAbsolute2.Busy OR stAxis.PTP.MoveAbsolute2.Done) THEN
			stAxis.PTP.MoveAbsolute1.Acceleration	:= 0;
			stAxis.PTP.MoveAbsolute1.BufferMode		:= MC_BlendingNext;
			stAxis.PTP.MoveAbsolute1.Deceleration	:= 0;
			stAxis.PTP.MoveAbsolute1.Execute		:= TRUE;
			stAxis.PTP.MoveAbsolute1.Jerk			:= 0;
			stAxis.PTP.MoveAbsolute1.Position		:= Axis.NcToPlc.ActPos + fConveyorLenght;
			stAxis.PTP.MoveAbsolute1.Velocity		:= PackTags.Command.Parameter[4].Value;
			stAxis.PTP.MoveAbsolute2.Execute		:= FALSE;
		ELSIF TrigbStartbelt.Q AND (stAxis.PTP.MoveAbsolute1.Busy OR stAxis.PTP.MoveAbsolute1.Done) THEN
			stAxis.PTP.MoveAbsolute2.Acceleration	:= 0;
			stAxis.PTP.MoveAbsolute2.BufferMode		:= MC_BlendingNext;
			stAxis.PTP.MoveAbsolute2.Deceleration	:= 0;
			stAxis.PTP.MoveAbsolute2.Execute		:= TRUE;
			stAxis.PTP.MoveAbsolute2.Jerk			:= 0;
			stAxis.PTP.MoveAbsolute2.Position		:= Axis.NcToPlc.ActPos + fConveyorLenght;
			stAxis.PTP.MoveAbsolute2.Velocity		:= PackTags.Command.Parameter[4].Value;
			stAxis.PTP.MoveAbsolute1.Execute		:= FALSE;
		ELSIF TrigbStartbelt.Q THEN
			stAxis.PTP.MoveAbsolute1.Acceleration	:= 0;
			stAxis.PTP.MoveAbsolute1.BufferMode		:= MC_BlendingNext;
			stAxis.PTP.MoveAbsolute1.Deceleration	:= 0;
			stAxis.PTP.MoveAbsolute1.Execute		:= TRUE;
			stAxis.PTP.MoveAbsolute1.Jerk			:= 0;
			stAxis.PTP.MoveAbsolute1.Position		:= Axis.NcToPlc.ActPos + fConveyorLenght;
			stAxis.PTP.MoveAbsolute1.Velocity		:= PackTags.Command.Parameter[4].Value;
			stAxis.PTP.MoveAbsolute2.Execute		:= FALSE;
		END_IF
		
		//Production target is reached
		IF	REAL_TO_DINT(PackTags.Command.Parameter[2].Value)	<= PackTags.Admin.ProdProcessedCount[1].Count
		  AND(NOT stAxis.PTP.MoveAbsolute1.Execute OR (NOT stAxis.PTP.MoveAbsolute1.Busy		AND  stAxis.PTP.MoveAbsolute1.Done))
		  AND(NOT stAxis.PTP.MoveAbsolute2.Execute OR (NOT stAxis.PTP.MoveAbsolute2.Busy		AND  stAxis.PTP.MoveAbsolute2.Done))
		  AND	AxisMain.Status.NotMoving						AND PackTags.Status.StateCurrent = ePMLState_Execute THEN
			stAxis.PTP.MoveAbsolute1.Execute		:= FALSE;
			stAxis.PTP.MoveAbsolute2.Execute		:= FALSE;
			M_StateComplete();
		END_IF
		
	ePMLProtUnitMode_Maintenance:
		//

	ePMLProtUnitMode_Manual:
		//Call FB_AxisGeneral
		SUPER^.M_Execute();

	ePMLUnitMode_Service:
		//
END_CASE
END_METHOD

{attribute 'object_name' := 'M_Holding'}
METHOD M_Holding
CASE fbUnitModeManager.eModeStatus OF	
	ePMLProtUnitMode_Production:	
		//Use two MoveAbsolute functionblocks, to use the Buffermode MC_BlendingNext
		IF TrigbStartbelt.Q AND (stAxis.PTP.MoveAbsolute2.Busy OR stAxis.PTP.MoveAbsolute2.Done) THEN
			stAxis.PTP.MoveAbsolute1.Acceleration	:= 0;
			stAxis.PTP.MoveAbsolute1.BufferMode		:= MC_BlendingNext;
			stAxis.PTP.MoveAbsolute1.Deceleration	:= 0;
			stAxis.PTP.MoveAbsolute1.Execute		:= TRUE;
			stAxis.PTP.MoveAbsolute1.Jerk			:= 0;
			stAxis.PTP.MoveAbsolute1.Position		:= Axis.NcToPlc.ActPos + fConveyorLenght;
			stAxis.PTP.MoveAbsolute1.Velocity		:= PackTags.Command.Parameter[4].Value;
			stAxis.PTP.MoveAbsolute2.Execute		:= FALSE;
		ELSIF TrigbStartbelt.Q AND (stAxis.PTP.MoveAbsolute1.Busy OR stAxis.PTP.MoveAbsolute1.Done) THEN
			stAxis.PTP.MoveAbsolute2.Acceleration	:= 0;
			stAxis.PTP.MoveAbsolute2.BufferMode		:= MC_BlendingNext;
			stAxis.PTP.MoveAbsolute2.Deceleration	:= 0;
			stAxis.PTP.MoveAbsolute2.Execute		:= TRUE;
			stAxis.PTP.MoveAbsolute2.Jerk			:= 0;
			stAxis.PTP.MoveAbsolute2.Position		:= Axis.NcToPlc.ActPos + fConveyorLenght;
			stAxis.PTP.MoveAbsolute2.Velocity		:= PackTags.Command.Parameter[4].Value;
			stAxis.PTP.MoveAbsolute1.Execute		:= FALSE;
		ELSIF TrigbStartbelt.Q THEN
			stAxis.PTP.MoveAbsolute1.Acceleration	:= 0;
			stAxis.PTP.MoveAbsolute1.BufferMode		:= MC_BlendingNext;
			stAxis.PTP.MoveAbsolute1.Deceleration	:= 0;
			stAxis.PTP.MoveAbsolute1.Execute		:= TRUE;
			stAxis.PTP.MoveAbsolute1.Jerk			:= 0;
			stAxis.PTP.MoveAbsolute1.Position		:= Axis.NcToPlc.ActPos + fConveyorLenght;
			stAxis.PTP.MoveAbsolute1.Velocity		:= PackTags.Command.Parameter[4].Value;
			stAxis.PTP.MoveAbsolute2.Execute		:= FALSE;
		END_IF
		
		IF AxisMain.Status.NotMoving AND NOT stAxis.PTP.MoveAbsolute1.Busy AND NOT stAxis.PTP.MoveAbsolute2.Busy THEN
			M_StateComplete();
		END_IF

	ePMLProtUnitMode_Maintenance:
		M_StateComplete();
END_CASE
END_METHOD

{attribute 'object_name' := 'M_Idle'}
METHOD M_Idle
iStateClearing	:= 0;
END_METHOD

{attribute 'object_name' := 'M_Resetting'}
METHOD M_Resetting
CASE fbStateMachine.eMode OF
	ePMLProtUnitMode_Production:	
		CASE iStateResetting OF
			0:
				//SW-Enable for the Axis
				bResettingDone										:= FALSE;
				stAxis.Admin.Power.BufferMode			:= MC_Aborting;
				stAxis.Admin.Power.Enable				:= TRUE;
				stAxis.Admin.Power.Enable_Negative		:= TRUE;
				stAxis.Admin.Power.Enable_Positive		:= TRUE;
				stAxis.Admin.Power.Override				:= 100.0;
				IF stAxis.Admin.Power.Status THEN
					iStateResetting	:= 1;
				END_IF
								
			1:
				//Take away all Motioncommands
				stAxis.PTP.Halt.Execute					:= FALSE;
				stAxis.PTP.MoveAbsolute1.Execute		:= FALSE;
				stAxis.PTP.MoveAbsolute2.Execute		:= FALSE;
				stAxis.PTP.MoveVelocitiy.Execute		:= FALSE;
				stAxis.PTP.Stop.Execute					:= FALSE;
				IF NOT Axis.Status.HasJob THEN
					iStateResetting									:= 2;
				END_IF
					
			2:
				//Move the Axis for one Conveyorroatation
				stAxis.PTP.MoveAbsolute1.Acceleration	:= 0;
				stAxis.PTP.MoveAbsolute1.BufferMode		:= MC_Aborting;
				stAxis.PTP.MoveAbsolute1.Deceleration	:= 0;
				stAxis.PTP.MoveAbsolute1.Execute		:= TRUE;
				stAxis.PTP.MoveAbsolute1.Jerk			:= 0;
				stAxis.PTP.MoveAbsolute1.Velocity		:= fConveyorVelo;
				stAxis.PTP.MoveAbsolute1.Position		:= (Axis.NcToPlc.ActPos + fConveyorLenght); //Drive actual Position + Length of Conveyor
				IF stAxis.PTP.MoveAbsolute1.Done  THEN
					bResettingDone								:= TRUE;
					iStateResetting							:= 3;
				END_IF
							
			3: 
				//Use two MoveAbsolute functionblocks, to use the Buffermode MC_BlendingNext
				IF TrigbStartbelt.Q AND (stAxis.PTP.MoveAbsolute2.Busy OR stAxis.PTP.MoveAbsolute2.Done) THEN
					stAxis.PTP.MoveAbsolute1.Acceleration	:= 0;
					stAxis.PTP.MoveAbsolute1.BufferMode		:= MC_BlendingNext;
					stAxis.PTP.MoveAbsolute1.Deceleration	:= 0;
					stAxis.PTP.MoveAbsolute1.Execute		:= TRUE;
					stAxis.PTP.MoveAbsolute1.Jerk			:= 0;
					stAxis.PTP.MoveAbsolute1.Position		:= Axis.NcToPlc.ActPos + fConveyorLenght;
					stAxis.PTP.MoveAbsolute1.Velocity		:= PackTags.Command.Parameter[4].Value;
					stAxis.PTP.MoveAbsolute2.Execute		:= FALSE;
				ELSIF TrigbStartbelt.Q AND (stAxis.PTP.MoveAbsolute1.Busy OR stAxis.PTP.MoveAbsolute1.Done) THEN
					stAxis.PTP.MoveAbsolute2.Acceleration	:= 0;
					stAxis.PTP.MoveAbsolute2.BufferMode		:= MC_BlendingNext;
					stAxis.PTP.MoveAbsolute2.Deceleration	:= 0;
					stAxis.PTP.MoveAbsolute2.Execute		:= TRUE;
					stAxis.PTP.MoveAbsolute2.Jerk			:= 0;
					stAxis.PTP.MoveAbsolute2.Position		:= Axis.NcToPlc.ActPos + fConveyorLenght;
					stAxis.PTP.MoveAbsolute2.Velocity		:= PackTags.Command.Parameter[4].Value;
					stAxis.PTP.MoveAbsolute1.Execute		:= FALSE;
				ELSIF TrigbStartbelt.Q THEN
					stAxis.PTP.MoveAbsolute1.Acceleration	:= 0;
					stAxis.PTP.MoveAbsolute1.BufferMode		:= MC_BlendingNext;
					stAxis.PTP.MoveAbsolute1.Deceleration	:= 0;
					stAxis.PTP.MoveAbsolute1.Execute		:= TRUE;
					stAxis.PTP.MoveAbsolute1.Jerk			:= 0;
					stAxis.PTP.MoveAbsolute1.Position		:= Axis.NcToPlc.ActPos + fConveyorLenght;
					stAxis.PTP.MoveAbsolute1.Velocity		:= PackTags.Command.Parameter[4].Value;
					stAxis.PTP.MoveAbsolute2.Execute		:= FALSE;
				END_IF
							
				IF bAxisMainResetDone THEN
					M_StateComplete();
				END_IF				
		END_CASE
		
	ePMLProtUnitMode_Maintenance, ePMLUnitMode_Service:
		M_StateComplete();

	ePMLProtUnitMode_Manual:
		//Call FB_AxisGeneral
		SUPER^.M_Resetting();
END_CASE
END_METHOD

{attribute 'object_name' := 'M_Suspending'}
METHOD M_Suspending
CASE fbUnitModeManager.eModeStatus OF
	ePMLProtUnitMode_Production:
		//Use two MoveAbsolute functionblocks, to use the Buffermode MC_BlendingNext. 
		IF TrigbStartbelt.Q AND (stAxis.PTP.MoveAbsolute2.Busy OR stAxis.PTP.MoveAbsolute2.Done) THEN
			stAxis.PTP.MoveAbsolute1.Acceleration	:= 0;
			stAxis.PTP.MoveAbsolute1.BufferMode		:= MC_BlendingNext;
			stAxis.PTP.MoveAbsolute1.Deceleration	:= 0;
			stAxis.PTP.MoveAbsolute1.Execute		:= TRUE;
			stAxis.PTP.MoveAbsolute1.Jerk			:= 0;
			stAxis.PTP.MoveAbsolute1.Position		:= Axis.NcToPlc.ActPos + fConveyorLenght;
			stAxis.PTP.MoveAbsolute1.Velocity		:= PackTags.Command.Parameter[4].Value;
			stAxis.PTP.MoveAbsolute2.Execute		:= FALSE;
		ELSIF TrigbStartbelt.Q AND (stAxis.PTP.MoveAbsolute1.Busy OR stAxis.PTP.MoveAbsolute1.Done) THEN
			stAxis.PTP.MoveAbsolute2.Acceleration	:= 0;
			stAxis.PTP.MoveAbsolute2.BufferMode		:= MC_BlendingNext;
			stAxis.PTP.MoveAbsolute2.Deceleration	:= 0;
			stAxis.PTP.MoveAbsolute2.Execute		:= TRUE;
			stAxis.PTP.MoveAbsolute2.Jerk			:= 0;
			stAxis.PTP.MoveAbsolute2.Position		:= Axis.NcToPlc.ActPos + fConveyorLenght;
			stAxis.PTP.MoveAbsolute2.Velocity		:= PackTags.Command.Parameter[4].Value;
			stAxis.PTP.MoveAbsolute1.Execute		:= FALSE;
		ELSIF TrigbStartbelt.Q THEN
			stAxis.PTP.MoveAbsolute1.Acceleration	:= 0;
			stAxis.PTP.MoveAbsolute1.BufferMode		:= MC_BlendingNext;
			stAxis.PTP.MoveAbsolute1.Deceleration	:= 0;
			stAxis.PTP.MoveAbsolute1.Execute		:= TRUE;
			stAxis.PTP.MoveAbsolute1.Jerk			:= 0;
			stAxis.PTP.MoveAbsolute1.Position		:= Axis.NcToPlc.ActPos + fConveyorLenght;
			stAxis.PTP.MoveAbsolute1.Velocity		:= PackTags.Command.Parameter[4].Value;
			stAxis.PTP.MoveAbsolute2.Execute		:= FALSE;
		END_IF
		
		IF AxisMain.Status.NotMoving AND NOT stAxis.PTP.MoveAbsolute1.Busy AND NOT stAxis.PTP.MoveAbsolute2.Busy THEN
			M_StateComplete();
		END_IF

	ePMLUnitMode_Service:
		M_StateComplete();
END_CASE
END_METHOD

{attribute 'object_name' := 'M_Undefined'}
METHOD M_Undefined
bUndefinedDone:= TRUE;
END_METHOD

END_FUNCTION_BLOCK

// ---- POUs/General/FB_Velocity.TcPOU
FUNCTION_BLOCK FB_Velocity
VAR_INPUT
	nActQuantity	: DINT;					//Number of finished products
END_VAR
VAR_OUTPUT
	fActVelocity	: REAL;					//Actual velocity 
	fAverageVelo	: REAL;					//Average Velocity
END_VAR
VAR
	fbTimer			: TON;
	aActQuantity	: ARRAY[0..6] OF DINT;	//Array to safe the last 6 Number of finished products
	aAverageVelo	: ARRAY[1..10] OF REAL;	//Array to safe the last 10 Velocities
	nCounting		: DINT ;				//Variable to runs step by step trough the array
END_VAR

fbTimer.PT	:= T#10S;
fbTimer.IN	:= TRUE;
IF fbTimer.Q THEN
	//calculate the current velocity, the measurement time is 60s, the Value is updating every 10s
	aActQuantity[6]	:= aActQuantity[5];
	aActQuantity[5]	:= aActQuantity[4];
	aActQuantity[4]	:= aActQuantity[3];
	aActQuantity[3]	:= aActQuantity[2];
	aActQuantity[2]	:= aActQuantity[1];
	aActQuantity[1]	:= aActQuantity[0];
	aActQuantity[0]	:= nActQuantity;
	
	fActVelocity :=DINT_TO_REAL( aActQuantity[0]-aActQuantity[6]) / (60.0/60.0);
	
	IF fActVelocity < 0 THEN
		fActVelocity	:= 0;
	END_IF

	//calculate the average velocity, the measurement time is 10*10s=100s, the value is updating every 10s
	FOR nCounting:=1 TO 9 BY 1 DO
		aAverageVelo[11-nCounting] := aAverageVelo[10-nCounting];
	END_FOR
	aAverageVelo[1] := fActVelocity;
	
	fAverageVelo		:= 0;
	FOR nCounting:=1 TO 10 BY 1 DO
		fAverageVelo	:= fAverageVelo + aAverageVelo[nCounting];
	END_FOR	
	fAverageVelo := fAverageVelo/10;
	
	fbTimer.IN	:= FALSE;
END_IF

IF PackTags.Status.StateCurrent = ePMLState_Complete OR stChangeIntoProduction.bYesReset THEN
	aActQuantity[6]	:= 0;
	aActQuantity[5]	:= 0;
	aActQuantity[4]	:= 0;
	aActQuantity[3]	:= 0;
	aActQuantity[2]	:= 0;
	aActQuantity[1]	:= 0;
	aActQuantity[0]	:= 0;
	fActVelocity	:= 0;
END_IF
fbTimer();

END_FUNCTION_BLOCK

// ---- POUs/General/FB_Visu.TcPOU
FUNCTION_BLOCK FB_Visu
VAR_INPUT
	// =============== Axis =====================================
	fAxisVelo						: LREAL;					// Axis velocity
	
	// =============== State of machine elements ================
	bMainAxisMoves					: BOOL;						// True if main axis is moving
	bMetalAxisMoves					: BOOL;						// True if metal axis is moving
	bPlasticAxisMoves				: BOOL;						// True if plastic axis is moving
	bClampToWork					: BOOL;						// True if clamp cylinder moves to work position
	bBarrierToWork					: BOOL;						// True if barrier cylinder moves to work position
	bMetalToWork					: BOOL;						// True if metal cylinder moves to work position
	bPlasticToWork					: BOOL;						// True if plastic cylinder moves to work position
	
	bReset							: BOOL;						// True if state machine is in state RESETTING
	
	// =============== Keys =====================================
	aKeyPressed						: ARRAY [1..12] OF BOOL;
	aUnitInfo						: ARRAY [1..12] OF ST_UnitInfo;
END_VAR
VAR_OUTPUT
	fYClamp							: LREAL;					// Y-Coordinate of clamp cylinder
	fYBarrier						: LREAL;					// Y-Coordinate of barrier cylinder
	fYMetal							: LREAL;					// Y-Coordinate of metal cylinder
	fYPlastic						: LREAL;					// Y-Coordinate of plastic cylinder
	
	// =============== Buttons of visualization - outputs =======
	bButtonPowerOut					: BOOL;						// To turn on and off the machine
	
	// Axis buttons
	bButtonMainFwOut				: BOOL;						// To move main axis forward
	bButtonMetalFwOut				: BOOL;						// To move metal axis forwards
	bButtonPlasticFwOut				: BOOL;						// To move plastic axis forwards
	
	// Cylinder buttons
	bButtonClampToWorkOut			: BOOL;						// To move manually clamp cylinder to work position
	bButtonBarrierToWorkOut			: BOOL;						// To move manually barrier cylinder to work position
	bButtonMetalToWorkOut			: BOOL;						// To move manually metal cylinder to work position
	bButtonPlasticToWorkOut			: BOOL;						// To move manually plastic cylinder to work position
	
	//=============== Cheking Button and entries =======================
	bInvalidEntry					: BOOL;						//Invalid entry, to produce products

	// =============== Keys =====================================
	aCaption						: ARRAY [1..12] OF STRING;	

	eModeVisu						: DINT;						// Mode for the 	StateChart	
	eStateVisu						: E_PMLState;				// State for the StateChart
	sUnitName						: STRING;
	iFrameVisible					: DINT;
END_VAR
VAR
	i								: DINT;
	
	// =============== Cylinder states ======================
	//The PlcTask Outputs(AT%Q*) are linked to the PlcTaks Inputs(AT%I*)
	bClampAtBase		AT %Q*		: BOOL;						// True if clamp cylinder is in base position
	bClampAtWork		AT %Q*		: BOOL;						// True if clamp cylinder is in work position
	bBarrierAtBase		AT %Q*		: BOOL;						// True if barrier cylinder is in base position
	bBarrierAtWork		AT %Q*		: BOOL;						// True if barrier cylinder is in work position
	bMetalAtBase		AT %Q*		: BOOL;						// True if metal cylinder is in base position
	bMetalAtWork		AT %Q*		: BOOL;						// True if metal cylinder is in work position
	bPlasticAtBase		AT %Q*		: BOOL;						// True if plastic cylinder is in base position
	bPlasticAtWork		AT %Q*		: BOOL;						// True if plastic cylinder is in work position

	// =============== Sensors to detect boxes ==============
	//The PlcTask Outputs(AT%Q*) are linked to the PlcTaks Inputs(AT%I*)
	bBarrierSensor		AT %Q*		: BOOL;						// True if barrier sensor detects a box
	bMetalSensor		AT %Q*		: BOOL;						// True if metal sensor detects a metal box
	bPlasticSensor		AT %Q*		: BOOL;						// True if plastic sensor detects a box

	// =============== Position variables ===================
	aBoxX							: ARRAY[1..4] OF LREAL;		// X-Coordinates of boxes
	aBoxY							: ARRAY[1..4] OF LREAL;		// Y-Coordinates of boxes
	
	// =============== Statechart variables ===================
	eUnitRepresentOnVisu			: E_UnitName := eMachine;	// Unit represent on Visu
		
	// =============== Warnings ===============================================
	sWarningVisu					: STRING;					// Descripton, name of the warning
	fbTimerWarning					: TON;						// Timer for visu textbox
	nWarningState					: INT :=0;					// State for representing warnings
	nWarningCount					: INT :=1;					// Variable to runs step by step trough the warningarray
	
	// =============== Errors ===============================================
	sAlarmVisu						: STRING;					// Descripton, name of the error
	fbTimerAlarm					: TON;						// Timer for visu textbox
	nAlarmState						: INT :=0;					// State for representing errors
	nAlarmCount						: INT :=1;					// Variable to runs step by step trough the errorarray
	
	// =============== Boxes movement ===========================
	nLastBox						: INT;						// Box on last position of main belt
	aBoxMetalMove					: ARRAY[1..4] OF BOOL;		// bBoxMetalMove[1] is true, if box 1 is moved by metal cylinder
	aBoxMetalFree					: ARRAY[1..4] OF BOOL;		// bBoxMetalFree[1] is true, if any box blockades the movement of box 1 on metal belt
	aBoxPlasticMove					: ARRAY[1..4] OF BOOL;		// bBoxPlasticMove[1] is true, if box 1 is moved by plastic cylinder
	aBoxPlasticFree					: ARRAY[1..4] OF BOOL;		// bBoxMetalFree[1] is true, if any box blockades the plastic belt
	aBoxMainBelt					: ARRAY[1..4] OF BOOL;		// bBoxMainBelt[1] is true, if box 1 is on main belt and has no obstacles, so box 1 is moved by main axis
	aBoxMetalBelt					: ARRAY[1..4] OF BOOL;		// aBoxMetalBelt[1] is true, if box 1 is on metal belt and has no obstacles, so box 1 is moved by metal axis
	aBoxPlasticBelt					: ARRAY[1..4] OF BOOL;		// aBoxPlasticBelt[1] is true, if box 1 is on plastic belt and has no obstacles, so box 1 is moved by plastic axis
	fMainVelo						: LREAL;					// Velocity of boxes on main belt
	fMetalVelo						: LREAL;					// Velocity of boxes on metal belt
	fPlasticVelo					: LREAL;					// Velocity of boxes on plastic belt
	bAccident						: BOOL;						// True if machine caused an accident
	nState							: INT;
	
	// =============== Axes movement ============================
	nAngleMain						: INT;						// Angle of main axis element
	nAngleMetal						: INT;						// Angle of metal axis element
	nAnglePlastic					: INT;						// Angle of plastic axis element
	fbTimerMainAxis					: TON;						// Timer for movement of main axis element
	fbTimerMetalAxis				: TON;						// Timer for movement of metal axis element
	fbTimerPlasticAxis				: TON;						// Timer for movement of plastic axis element
	tMoveAxis						: TIME := T#40MS;			// Time for movement of elements

	
	nButtonColorClamp				: DWORD;					// Color of button to move clamp cylinder
	bButtonColorClamp				: BOOL;						// To change color of clamp button
	nButtonColorBarrier				: DWORD;					// Color of button to move barrier cylinder
	bButtonColorBarrier				: BOOL;						// To change color of barrier button
	nButtonColorMetalCyl			: DWORD;					// Color of button to move metal cylinder
	bButtonColorMetalCyl			: BOOL;						// To change color of metal cylinder button
	nButtonColorPlasticCyl			: DWORD;					// Color of button to move plastic cylinder
	bButtonColorPlasticCyl			: BOOL;						// To change color of plastic cylinder button
	nButtonColorMainFw				: DWORD;					// Color of button to move main axis forwards
	bButtonColorMainFw				: BOOL;						// To change color of button to move main axis fw.
	nButtonColorMetalFw				: DWORD;					// Color of button to move metal axis forwards
	bButtonColorMetalFw				: BOOL;						// To change color of button to move metal axis fw.
	nButtonColorPlasticFw			: DWORD;					// Color of button to move plastic axis forwards
	bButtonColorPlasticFw			: BOOL;						// To change color of button to move plastic axis fw.
END_VAR
VAR CONSTANT	
	// =============== Velocities ===========================================
	cVelocityDenominator						: LREAL := 250.0;			// Velocity of visualization is a fraction of real axis velocity
	cAxisMovementSemiPlusAuto					: INT 	:= 2;				// Axis movement per cycle in mode Automatic and Semi Autoamtic
	cAxisMovementManual							: INT 	:= 1;				// Axis movement per cycle in mode Manual
	cClampMovement								: LREAL := 0.1;				// Cylinder movement per cycle for clamp cylinder
	cBarrierMovement							: LREAL := 1.0;				// Cylinder movement per cycle for barrier cylinder
	cMetalPlasticCylMovement					: LREAL := 1.0;				// Cylinder movement per cycle for metal and plastic cylinder
	
	// =============== Barrier, clamp, metal, plastic cylinder ==============
	cYClampCylStartPos							: LREAL := 0.0;				// Y-start-position of clamp cylinder (where movement starts)
	cYClampCylEndPos							: LREAL := 3.0;				// Y-end-position of clamp cylinder (where movement ends)
	cYBarrierCylStartPos						: LREAL := 0.0;				// Y-start-position of barrier cylinder (where movement starts)
	cYBarrierCylEndPos							: LREAL := 63.0;			// Y-end-position of barrier cylinder (where movement ends)
	cYMetalPlasticCylStartPos					: LREAL := 0.0;				// Y-start-position of metal and plastic cylinder (where movement starts)
	cYMetalPlasticCylEndPos						: LREAL := -73.0;			// Y-end-position of metal and plastic cylinder (where movement ends)
	
	// =============== Widths, distances ====================================
	cBoxWidth									: LREAL := 60.0;			// Width of a box in the visu
	cBarrierWidth								: LREAL := 30.0;			// Width of the barrier cylinder in the visu
	cDiffBarrierToStartOfMetalCyl				: LREAL := 191.0;			// Difference on visu from barrier to start of metal cylinder
	cDiffBarrierToEndOfMetalCyl					: LREAL := 261.0;			// Difference on visu from barrier to end of metal cylinder
	cDiffBarrierToStartOfPlasticCyl				: LREAL := 441.0;			// Difference on visu from barrier to start of plastic cylinder
	cYMetalPlasticCylOnMainBelt					: LREAL := -9.0;			// Y-Position of metal and plastic cylinder reaching the main belt
	cYBoxesOnMetalPlasticBelt_min				: LREAL := -65.0;			// Minimal Y-Position of boxes when being on metal or plastic belt
	cYBoxesOnMetalPlasticBelt_max				: LREAL := -140.0;			// Maximal Y-Position of boxes when being on metal or plastic belt
	
	// =============== Positions of boxes - main belt =======================
	cYforAllBoxesOnMainBelt						: LREAL := -5.0;			// Y-Position of boxes being on main belt
	cYforAllBoxesNotOnMainBelt					: LREAL := -60.0;			// Y-Position of boxes not being on main belt
	
	cYforAllBoxesStartPosMainBelt				: LREAL := 0.0;				// Y-Position of boxes when being on first position of main belt
	cXforAllBoxesStartPosMainBelt				: LREAL := -240.0;			// X-Position of boxes when being on first position of main belt
	cXforAllBoxesLastPossiblePosMainBelt		: LREAL := 461.0;			// Last possible X-position of boxes on main belt
	
	cXforAllBoxesCorrectPushMetalCyl_min		: LREAL := 180;				// Minimal X-Position of boxes when being pushed by metal cylinder to metal belt 
	cXforAllBoxesCorrectPushMetalCyl_max		: LREAL := 211;				// Maximal X-Position of boxes when being pushed by metal cylinder to metal belt 
	cXforAllBoxesIncorrectPushMetalCyl_min		: LREAL := 131;				// Minimal X-Position of boxes when being pushed by metal cylinder, but not pushed to metal belt
	cXforAllBoxesIncorrectPushMetalCyl_max		: LREAL := 261;				// Maximal X-Position of boxes when being pushed by metal cylinder, but not pushed to metal belt
	
	cXforAllBoxesCorrectPushPlasticCyl_min		: LREAL := 430;				// Minimal X-Position of boxes when being pushed by plastic cylinder to plastic belt 
	cXforAllBoxesCorrectPushPlasticCyl_max		: LREAL := 461;				// Minimal X-Position of boxes when being pushed by plastic cylinder to plastic belt 
	cXforAllBoxesIncorrectPushPlasticCyl_min	: LREAL := 381;				// Minimal X-Position of boxes when being pushed by plastic cylinder, but not pushed to plastic belt
	
